    GB2312[3982]:= 16#f1b6;
    GB2312[3983]:= 16#f1b7;
    GB2312[3984]:= 16#bfd5;
    GB2312[3985]:= 16#b4a9;
    GB2312[3986]:= 16#f1b8;
    GB2312[3987]:= 16#cdbb;
    GB2312[3988]:= 16#c7d4;
    GB2312[3989]:= 16#d5ad;
    GB2312[3990]:= 16#f1b9;
    GB2312[3991]:= 16#f1ba;
    GB2312[3992]:= 16#c7cf;
    GB2312[3993]:= 16#d2a4;
    GB2312[3994]:= 16#d6cf;
    GB2312[3995]:= 16#f1bb;
    GB2312[3996]:= 16#bdd1;
    GB2312[3997]:= 16#b4b0;
    GB2312[3998]:= 16#bebd;
    GB2312[3999]:= 16#b4dc;              //GB2312码 3000-3999
END_IF;
(* Rung 15 *)
IF P_On THEN
    GB2312[4000]:= 16#ced1;
    GB2312[4001]:= 16#bfdf;
    GB2312[4002]:= 16#f1bd;
    GB2312[4003]:= 16#bffa;
    GB2312[4004]:= 16#f1bc;
    GB2312[4005]:= 16#f1bf;
    GB2312[4006]:= 16#f1be;
    GB2312[4007]:= 16#f1c0;
    GB2312[4008]:= 16#f1c1;
    GB2312[4009]:= 16#c1fe;
    GB2312[4010]:= 16#c1a2;
    GB2312[4011]:= 16#cafa;
    GB2312[4012]:= 16#d5be;
    GB2312[4013]:= 16#beba;
    GB2312[4014]:= 16#beb9;
    GB2312[4015]:= 16#d5c2;
    GB2312[4016]:= 16#bfa2;
    GB2312[4017]:= 16#cdaf;
    GB2312[4018]:= 16#f1b5;
    GB2312[4019]:= 16#bddf;
    GB2312[4020]:= 16#b6cb;
    GB2312[4021]:= 16#d6f1;
    GB2312[4022]:= 16#f3c3;
    GB2312[4023]:= 16#f3c4;
    GB2312[4024]:= 16#b8cd;
    GB2312[4025]:= 16#f3c6;
    GB2312[4026]:= 16#f3c7;
    GB2312[4027]:= 16#b0ca;
    GB2312[4028]:= 16#f3c5;
    GB2312[4029]:= 16#f3c9;
    GB2312[4030]:= 16#cbf1;
    GB2312[4031]:= 16#f3cb;
    GB2312[4032]:= 16#d0a6;
    GB2312[4033]:= 16#b1ca;
    GB2312[4034]:= 16#f3c8;
    GB2312[4035]:= 16#f3cf;
    GB2312[4036]:= 16#b5d1;
    GB2312[4037]:= 16#f3d7;
    GB2312[4038]:= 16#f3d2;
    GB2312[4039]:= 16#f3d4;
    GB2312[4040]:= 16#f3d3;
    GB2312[4041]:= 16#b7fb;
    GB2312[4042]:= 16#b1bf;
    GB2312[4043]:= 16#f3ce;
    GB2312[4044]:= 16#f3ca;
    GB2312[4045]:= 16#b5da;
    GB2312[4046]:= 16#f3d0;
    GB2312[4047]:= 16#f3d1;
    GB2312[4048]:= 16#f3d5;
    GB2312[4049]:= 16#f3cd;
    GB2312[4050]:= 16#bce3;
    GB2312[4051]:= 16#c1fd;
    GB2312[4052]:= 16#f3d6;
    GB2312[4053]:= 16#f3da;
    GB2312[4054]:= 16#f3cc;
    GB2312[4055]:= 16#b5c8;
    GB2312[4056]:= 16#bdee;
    GB2312[4057]:= 16#f3dc;
    GB2312[4058]:= 16#b7a4;
    GB2312[4059]:= 16#bff0;
    GB2312[4060]:= 16#d6fe;
    GB2312[4061]:= 16#cdb2;
    GB2312[4062]:= 16#b4f0;
    GB2312[4063]:= 16#b2df;
    GB2312[4064]:= 16#f3d8;
    GB2312[4065]:= 16#f3d9;
    GB2312[4066]:= 16#c9b8;
    GB2312[4067]:= 16#f3dd;
    GB2312[4068]:= 16#f3de;
    GB2312[4069]:= 16#f3e1;
    GB2312[4070]:= 16#f3df;
    GB2312[4071]:= 16#f3e3;
    GB2312[4072]:= 16#f3e2;
    GB2312[4073]:= 16#f3db;
    GB2312[4074]:= 16#bfea;
    GB2312[4075]:= 16#b3ef;
    GB2312[4076]:= 16#f3e0;
    GB2312[4077]:= 16#c7a9;
    GB2312[4078]:= 16#bcf2;
    GB2312[4079]:= 16#f3eb;
    GB2312[4080]:= 16#b9bf;
    GB2312[4081]:= 16#f3e4;
    GB2312[4082]:= 16#b2ad;
    GB2312[4083]:= 16#bbfe;
    GB2312[4084]:= 16#cbe3;
    GB2312[4085]:= 16#f3ed;
    GB2312[4086]:= 16#f3e9;
    GB2312[4087]:= 16#b9dc;
    GB2312[4088]:= 16#f3ee;
    GB2312[4089]:= 16#f3e5;
    GB2312[4090]:= 16#f3e6;
    GB2312[4091]:= 16#f3ea;
    GB2312[4092]:= 16#c2e1;
    GB2312[4093]:= 16#f3ec;
    GB2312[4094]:= 16#f3ef;
    GB2312[4095]:= 16#f3e8;
    GB2312[4096]:= 16#bcfd;
    GB2312[4097]:= 16#cfe4;
    GB2312[4098]:= 16#f3f0;
    GB2312[4099]:= 16#f3e7;
    GB2312[4100]:= 16#f3f2;
    GB2312[4101]:= 16#d7ad;
    GB2312[4102]:= 16#c6aa;
    GB2312[4103]:= 16#f3f3;
    GB2312[4104]:= 16#f3f1;
    GB2312[4105]:= 16#c2a8;
    GB2312[4106]:= 16#b8dd;
    GB2312[4107]:= 16#f3f5;
    GB2312[4108]:= 16#f3f4;
    GB2312[4109]:= 16#b4db;
    GB2312[4110]:= 16#f3f6;
    GB2312[4111]:= 16#f3f7;
    GB2312[4112]:= 16#f3f8;
    GB2312[4113]:= 16#c0ba;
    GB2312[4114]:= 16#c0e9;
    GB2312[4115]:= 16#c5f1;
    GB2312[4116]:= 16#f3fb;
    GB2312[4117]:= 16#f3fa;
    GB2312[4118]:= 16#b4d8;
    GB2312[4119]:= 16#f3fe;
    GB2312[4120]:= 16#f3f9;
    GB2312[4121]:= 16#f3fc;
    GB2312[4122]:= 16#f3fd;
    GB2312[4123]:= 16#f4a1;
    GB2312[4124]:= 16#f4a3;
    GB2312[4125]:= 16#bbc9;
    GB2312[4126]:= 16#f4a2;
    GB2312[4127]:= 16#f4a4;
    GB2312[4128]:= 16#b2be;
    GB2312[4129]:= 16#f4a6;
    GB2312[4130]:= 16#f4a5;
    GB2312[4131]:= 16#bcae;
    GB2312[4132]:= 16#c3d7;
    GB2312[4133]:= 16#d9e1;
    GB2312[4134]:= 16#c0e0;
    GB2312[4135]:= 16#f4cc;
    GB2312[4136]:= 16#d7d1;
    GB2312[4137]:= 16#b7db;
    GB2312[4138]:= 16#f4ce;
    GB2312[4139]:= 16#c1a3;
    GB2312[4140]:= 16#c6c9;
    GB2312[4141]:= 16#b4d6;
    GB2312[4142]:= 16#d5b3;
    GB2312[4143]:= 16#f4d0;
    GB2312[4144]:= 16#f4cf;
    GB2312[4145]:= 16#f4d1;
    GB2312[4146]:= 16#cbda;
    GB2312[4147]:= 16#f4d2;
    GB2312[4148]:= 16#d4c1;
    GB2312[4149]:= 16#d6e0;
    GB2312[4150]:= 16#b7e0;
    GB2312[4151]:= 16#c1b8;
    GB2312[4152]:= 16#c1bb;
    GB2312[4153]:= 16#f4d3;
    GB2312[4154]:= 16#beac;
    GB2312[4155]:= 16#b4e2;
    GB2312[4156]:= 16#f4d4;
    GB2312[4157]:= 16#f4d5;
    GB2312[4158]:= 16#beab;
    GB2312[4159]:= 16#f4d6;
    GB2312[4160]:= 16#f4db;
    GB2312[4161]:= 16#f4d7;
    GB2312[4162]:= 16#f4da;
    GB2312[4163]:= 16#bafd;
    GB2312[4164]:= 16#f4d8;
    GB2312[4165]:= 16#f4d9;
    GB2312[4166]:= 16#b8e2;
    GB2312[4167]:= 16#ccc7;
    GB2312[4168]:= 16#f4dc;
    GB2312[4169]:= 16#b2da;
    GB2312[4170]:= 16#c3d3;
    GB2312[4171]:= 16#d4e3;
    GB2312[4172]:= 16#bfb7;
    GB2312[4173]:= 16#f4dd;
    GB2312[4174]:= 16#c5b4;
    GB2312[4175]:= 16#f4e9;
    GB2312[4176]:= 16#cfb5;
    GB2312[4177]:= 16#cec9;
    GB2312[4178]:= 16#cbd8;
    GB2312[4179]:= 16#cbf7;
    GB2312[4180]:= 16#bdf4;
    GB2312[4181]:= 16#d7cf;
    GB2312[4182]:= 16#c0db;
    GB2312[4183]:= 16#d0f5;
    GB2312[4184]:= 16#f4ea;
    GB2312[4185]:= 16#f4eb;
    GB2312[4186]:= 16#f4ec;
    GB2312[4187]:= 16#f7e3;
    GB2312[4188]:= 16#b7b1;
    GB2312[4189]:= 16#f4ed;
    GB2312[4190]:= 16#d7eb;
    GB2312[4191]:= 16#f4ee;
    GB2312[4192]:= 16#e6f9;
    GB2312[4193]:= 16#bec0;
    GB2312[4194]:= 16#e6fa;
    GB2312[4195]:= 16#baec;
    GB2312[4196]:= 16#e6fb;
    GB2312[4197]:= 16#cfcb;
    GB2312[4198]:= 16#e6fc;
    GB2312[4199]:= 16#d4bc;
    GB2312[4200]:= 16#bcb6;
    GB2312[4201]:= 16#e6fd;
    GB2312[4202]:= 16#e6fe;
    GB2312[4203]:= 16#bccd;
    GB2312[4204]:= 16#c8d2;
    GB2312[4205]:= 16#ceb3;
    GB2312[4206]:= 16#e7a1;
    GB2312[4207]:= 16#b4bf;
    GB2312[4208]:= 16#e7a2;
    GB2312[4209]:= 16#c9b4;
    GB2312[4210]:= 16#b8d9;
    GB2312[4211]:= 16#c4c9;
    GB2312[4212]:= 16#d7dd;
    GB2312[4213]:= 16#c2da;
    GB2312[4214]:= 16#b7d7;
    GB2312[4215]:= 16#d6bd;
    GB2312[4216]:= 16#cec6;
    GB2312[4217]:= 16#b7c4;
    GB2312[4218]:= 16#c5a6;
    GB2312[4219]:= 16#e7a3;
    GB2312[4220]:= 16#cfdf;
    GB2312[4221]:= 16#e7a4;
    GB2312[4222]:= 16#e7a5;
    GB2312[4223]:= 16#e7a6;
    GB2312[4224]:= 16#c1b7;
    GB2312[4225]:= 16#d7e9;
    GB2312[4226]:= 16#c9f0;
    GB2312[4227]:= 16#cfb8;
    GB2312[4228]:= 16#d6af;
    GB2312[4229]:= 16#d6d5;
    GB2312[4230]:= 16#e7a7;
    GB2312[4231]:= 16#b0ed;
    GB2312[4232]:= 16#e7a8;
    GB2312[4233]:= 16#e7a9;
    GB2312[4234]:= 16#c9dc;
    GB2312[4235]:= 16#d2ef;
    GB2312[4236]:= 16#bead;
    GB2312[4237]:= 16#e7aa;
    GB2312[4238]:= 16#b0f3;
    GB2312[4239]:= 16#c8de;
    GB2312[4240]:= 16#bde1;
    GB2312[4241]:= 16#e7ab;
    GB2312[4242]:= 16#c8c6;
    GB2312[4243]:= 16#e7ac;
    GB2312[4244]:= 16#bbe6;
    GB2312[4245]:= 16#b8f8;
    GB2312[4246]:= 16#d1a4;
    GB2312[4247]:= 16#e7ad;
    GB2312[4248]:= 16#c2e7;
    GB2312[4249]:= 16#bef8;
    GB2312[4250]:= 16#bdca;
    GB2312[4251]:= 16#cdb3;
    GB2312[4252]:= 16#e7ae;
    GB2312[4253]:= 16#e7af;
    GB2312[4254]:= 16#beee;
    GB2312[4255]:= 16#d0e5;
    GB2312[4256]:= 16#cbe7;
    GB2312[4257]:= 16#ccd0;
    GB2312[4258]:= 16#bccc;
    GB2312[4259]:= 16#e7b0;
    GB2312[4260]:= 16#bca8;
    GB2312[4261]:= 16#d0f7;
    GB2312[4262]:= 16#e7b1;
    GB2312[4263]:= 16#d0f8;
    GB2312[4264]:= 16#e7b2;
    GB2312[4265]:= 16#e7b3;
    GB2312[4266]:= 16#b4c2;
    GB2312[4267]:= 16#e7b4;
    GB2312[4268]:= 16#e7b5;
    GB2312[4269]:= 16#c9fe;
    GB2312[4270]:= 16#ceac;
    GB2312[4271]:= 16#c3e0;
    GB2312[4272]:= 16#e7b7;
    GB2312[4273]:= 16#b1c1;
    GB2312[4274]:= 16#b3f1;
    GB2312[4275]:= 16#e7b8;
    GB2312[4276]:= 16#e7b9;
    GB2312[4277]:= 16#d7db;
    GB2312[4278]:= 16#d5c0;
    GB2312[4279]:= 16#e7ba;
    GB2312[4280]:= 16#c2cc;
    GB2312[4281]:= 16#d7ba;
    GB2312[4282]:= 16#e7bb;
    GB2312[4283]:= 16#e7bc;
    GB2312[4284]:= 16#e7bd;
    GB2312[4285]:= 16#bcea;
    GB2312[4286]:= 16#c3e5;
    GB2312[4287]:= 16#c0c2;
    GB2312[4288]:= 16#e7be;
    GB2312[4289]:= 16#e7bf;
    GB2312[4290]:= 16#bca9;
    GB2312[4291]:= 16#e7c0;
    GB2312[4292]:= 16#e7c1;
    GB2312[4293]:= 16#e7b6;
    GB2312[4294]:= 16#b6d0;
    GB2312[4295]:= 16#e7c2;
    GB2312[4296]:= 16#e7c3;
    GB2312[4297]:= 16#e7c4;
    GB2312[4298]:= 16#bbba;
    GB2312[4299]:= 16#b5de;
    GB2312[4300]:= 16#c2c6;
    GB2312[4301]:= 16#b1e0;
    GB2312[4302]:= 16#e7c5;
    GB2312[4303]:= 16#d4b5;
    GB2312[4304]:= 16#e7c6;
    GB2312[4305]:= 16#b8bf;
    GB2312[4306]:= 16#e7c8;
    GB2312[4307]:= 16#e7c7;
    GB2312[4308]:= 16#b7ec;
    GB2312[4309]:= 16#e7c9;
    GB2312[4310]:= 16#b2f8;
    GB2312[4311]:= 16#e7ca;
    GB2312[4312]:= 16#e7cb;
    GB2312[4313]:= 16#e7cc;
    GB2312[4314]:= 16#e7cd;
    GB2312[4315]:= 16#e7ce;
    GB2312[4316]:= 16#e7cf;
    GB2312[4317]:= 16#e7d0;
    GB2312[4318]:= 16#d3a7;
    GB2312[4319]:= 16#cbf5;
    GB2312[4320]:= 16#e7d1;
    GB2312[4321]:= 16#e7d2;
    GB2312[4322]:= 16#e7d3;
    GB2312[4323]:= 16#e7d4;
    GB2312[4324]:= 16#c9c9;
    GB2312[4325]:= 16#e7d5;
    GB2312[4326]:= 16#e7d6;
    GB2312[4327]:= 16#e7d7;
    GB2312[4328]:= 16#e7d8;
    GB2312[4329]:= 16#e7d9;
    GB2312[4330]:= 16#bdc9;
    GB2312[4331]:= 16#e7da;
    GB2312[4332]:= 16#f3be;
    GB2312[4333]:= 16#b8d7;
    GB2312[4334]:= 16#c8b1;
    GB2312[4335]:= 16#f3bf;
    GB2312[4336]:= 16#f3c0;
    GB2312[4337]:= 16#f3c1;
    GB2312[4338]:= 16#b9de;
    GB2312[4339]:= 16#cdf8;
    GB2312[4340]:= 16#d8e8;
    GB2312[4341]:= 16#bab1;
    GB2312[4342]:= 16#c2de;
    GB2312[4343]:= 16#eeb7;
    GB2312[4344]:= 16#b7a3;
    GB2312[4345]:= 16#eeb9;
    GB2312[4346]:= 16#eeb8;
    GB2312[4347]:= 16#b0d5;
    GB2312[4348]:= 16#eebb;
    GB2312[4349]:= 16#d5d6;
    GB2312[4350]:= 16#d7ef;
    GB2312[4351]:= 16#d6c3;
    GB2312[4352]:= 16#eebd;
    GB2312[4353]:= 16#caf0;
    GB2312[4354]:= 16#eebc;
    GB2312[4355]:= 16#eebe;
    GB2312[4356]:= 16#eec0;
    GB2312[4357]:= 16#eebf;
    GB2312[4358]:= 16#d1f2;
    GB2312[4359]:= 16#c7bc;
    GB2312[4360]:= 16#c3c0;
    GB2312[4361]:= 16#b8e1;
    GB2312[4362]:= 16#c1e7;
    GB2312[4363]:= 16#f4c6;
    GB2312[4364]:= 16#d0df;
    GB2312[4365]:= 16#f4c7;
    GB2312[4366]:= 16#cfdb;
    GB2312[4367]:= 16#c8ba;
    GB2312[4368]:= 16#f4c8;
    GB2312[4369]:= 16#f4c9;
    GB2312[4370]:= 16#f4ca;
    GB2312[4371]:= 16#f4cb;
    GB2312[4372]:= 16#d9fa;
    GB2312[4373]:= 16#b8fe;
    GB2312[4374]:= 16#e5f1;
    GB2312[4375]:= 16#d3f0;
    GB2312[4376]:= 16#f4e0;
    GB2312[4377]:= 16#cecc;
    GB2312[4378]:= 16#b3e1;
    GB2312[4379]:= 16#f1b4;
    GB2312[4380]:= 16#d2ee;
    GB2312[4381]:= 16#f4e1;
    GB2312[4382]:= 16#cfe8;
    GB2312[4383]:= 16#f4e2;
    GB2312[4384]:= 16#c7cc;
    GB2312[4385]:= 16#b5d4;
    GB2312[4386]:= 16#b4e4;
    GB2312[4387]:= 16#f4e4;
    GB2312[4388]:= 16#f4e3;
    GB2312[4389]:= 16#f4e5;
    GB2312[4390]:= 16#f4e6;
    GB2312[4391]:= 16#f4e7;
    GB2312[4392]:= 16#bab2;
    GB2312[4393]:= 16#b0bf;
    GB2312[4394]:= 16#f4e8;
    GB2312[4395]:= 16#b7ad;
    GB2312[4396]:= 16#d2ed;
    GB2312[4397]:= 16#d2ab;
    GB2312[4398]:= 16#c0cf;
    GB2312[4399]:= 16#bfbc;
    GB2312[4400]:= 16#eba3;
    GB2312[4401]:= 16#d5df;
    GB2312[4402]:= 16#eac8;
    GB2312[4403]:= 16#f1f3;
    GB2312[4404]:= 16#b6f8;
    GB2312[4405]:= 16#cba3;
    GB2312[4406]:= 16#c4cd;
    GB2312[4407]:= 16#f1e7;
    GB2312[4408]:= 16#f1e8;
    GB2312[4409]:= 16#b8fb;
    GB2312[4410]:= 16#f1e9;
    GB2312[4411]:= 16#bac4;
    GB2312[4412]:= 16#d4c5;
    GB2312[4413]:= 16#b0d2;
    GB2312[4414]:= 16#f1ea;
    GB2312[4415]:= 16#f1eb;
    GB2312[4416]:= 16#f1ec;
    GB2312[4417]:= 16#f1ed;
    GB2312[4418]:= 16#f1ee;
    GB2312[4419]:= 16#f1ef;
    GB2312[4420]:= 16#f1f1;
    GB2312[4421]:= 16#f1f0;
    GB2312[4422]:= 16#c5d5;
    GB2312[4423]:= 16#f1f2;
    GB2312[4424]:= 16#b6fa;
    GB2312[4425]:= 16#f1f4;
    GB2312[4426]:= 16#d2ae;
    GB2312[4427]:= 16#dec7;
    GB2312[4428]:= 16#cbca;
    GB2312[4429]:= 16#b3dc;
    GB2312[4430]:= 16#b5a2;
    GB2312[4431]:= 16#b9a2;
    GB2312[4432]:= 16#c4f4;
    GB2312[4433]:= 16#f1f5;
    GB2312[4434]:= 16#f1f6;
    GB2312[4435]:= 16#c1c4;
    GB2312[4436]:= 16#c1fb;
    GB2312[4437]:= 16#d6b0;
    GB2312[4438]:= 16#f1f7;
    GB2312[4439]:= 16#f1f8;
    GB2312[4440]:= 16#c1aa;
    GB2312[4441]:= 16#c6b8;
    GB2312[4442]:= 16#bedb;
    GB2312[4443]:= 16#f1f9;
    GB2312[4444]:= 16#b4cf;
    GB2312[4445]:= 16#f1fa;
    GB2312[4446]:= 16#edb2;
    GB2312[4447]:= 16#edb1;
    GB2312[4448]:= 16#cbe0;
    GB2312[4449]:= 16#d2de;
    GB2312[4450]:= 16#cbc1;
    GB2312[4451]:= 16#d5d8;
    GB2312[4452]:= 16#c8e2;
    GB2312[4453]:= 16#c0df;
    GB2312[4454]:= 16#bca1;
    GB2312[4455]:= 16#ebc1;
    GB2312[4456]:= 16#d0a4;
    GB2312[4457]:= 16#d6e2;
    GB2312[4458]:= 16#b6c7;
    GB2312[4459]:= 16#b8d8;
    GB2312[4460]:= 16#ebc0;
    GB2312[4461]:= 16#b8ce;
    GB2312[4462]:= 16#ebbf;
    GB2312[4463]:= 16#b3a6;
    GB2312[4464]:= 16#b9c9;
    GB2312[4465]:= 16#d6ab;
    GB2312[4466]:= 16#b7f4;
    GB2312[4467]:= 16#b7ca;
    GB2312[4468]:= 16#bce7;
    GB2312[4469]:= 16#b7be;
    GB2312[4470]:= 16#ebc6;
    GB2312[4471]:= 16#ebc7;
    GB2312[4472]:= 16#b0b9;
    GB2312[4473]:= 16#bfcf;
    GB2312[4474]:= 16#ebc5;
    GB2312[4475]:= 16#d3fd;
    GB2312[4476]:= 16#ebc8;
    GB2312[4477]:= 16#ebc9;
    GB2312[4478]:= 16#b7ce;
    GB2312[4479]:= 16#ebc2;
    GB2312[4480]:= 16#ebc4;
    GB2312[4481]:= 16#c9f6;
    GB2312[4482]:= 16#d6d7;
    GB2312[4483]:= 16#d5cd;
    GB2312[4484]:= 16#d0b2;
    GB2312[4485]:= 16#ebcf;
    GB2312[4486]:= 16#ceb8;
    GB2312[4487]:= 16#ebd0;
    GB2312[4488]:= 16#b5a8;
    GB2312[4489]:= 16#b1b3;
    GB2312[4490]:= 16#ebd2;
    GB2312[4491]:= 16#cca5;
    GB2312[4492]:= 16#c5d6;
    GB2312[4493]:= 16#ebd3;
    GB2312[4494]:= 16#ebd1;
    GB2312[4495]:= 16#c5df;
    GB2312[4496]:= 16#ebce;
    GB2312[4497]:= 16#caa4;
    GB2312[4498]:= 16#ebd5;
    GB2312[4499]:= 16#b0fb;
    GB2312[4500]:= 16#bafa;
    GB2312[4501]:= 16#d8b7;
    GB2312[4502]:= 16#f1e3;
    GB2312[4503]:= 16#ebca;
    GB2312[4504]:= 16#ebcb;
    GB2312[4505]:= 16#ebcc;
    GB2312[4506]:= 16#ebcd;
    GB2312[4507]:= 16#ebd6;
    GB2312[4508]:= 16#e6c0;
    GB2312[4509]:= 16#ebd9;
    GB2312[4510]:= 16#bfe8;
    GB2312[4511]:= 16#d2c8;
    GB2312[4512]:= 16#ebd7;
    GB2312[4513]:= 16#ebdc;
    GB2312[4514]:= 16#b8ec;
    GB2312[4515]:= 16#ebd8;
    GB2312[4516]:= 16#bdba;
    GB2312[4517]:= 16#d0d8;
    GB2312[4518]:= 16#b0b7;
    GB2312[4519]:= 16#ebdd;
    GB2312[4520]:= 16#c4dc;
    GB2312[4521]:= 16#d6ac;
    GB2312[4522]:= 16#b4e0;
    GB2312[4523]:= 16#c2f6;
    GB2312[4524]:= 16#bcb9;
    GB2312[4525]:= 16#ebda;
    GB2312[4526]:= 16#ebdb;
    GB2312[4527]:= 16#d4e0;
    GB2312[4528]:= 16#c6ea;
    GB2312[4529]:= 16#c4d4;
    GB2312[4530]:= 16#ebdf;
    GB2312[4531]:= 16#c5a7;
    GB2312[4532]:= 16#d9f5;
    GB2312[4533]:= 16#b2b1;
    GB2312[4534]:= 16#ebe4;
    GB2312[4535]:= 16#bdc5;
    GB2312[4536]:= 16#ebe2;
    GB2312[4537]:= 16#ebe3;
    GB2312[4538]:= 16#b8ac;
    GB2312[4539]:= 16#cdd1;
    GB2312[4540]:= 16#ebe5;
    GB2312[4541]:= 16#ebe1;
    GB2312[4542]:= 16#c1b3;
    GB2312[4543]:= 16#c6a2;
    GB2312[4544]:= 16#ccf3;
    GB2312[4545]:= 16#ebe6;
    GB2312[4546]:= 16#c0b0;
    GB2312[4547]:= 16#d2b8;
    GB2312[4548]:= 16#ebe7;
    GB2312[4549]:= 16#b8af;
    GB2312[4550]:= 16#b8ad;
    GB2312[4551]:= 16#ebe8;
    GB2312[4552]:= 16#c7bb;
    GB2312[4553]:= 16#cdf3;
    GB2312[4554]:= 16#ebea;
    GB2312[4555]:= 16#ebeb;
    GB2312[4556]:= 16#ebed;
    GB2312[4557]:= 16#d0c8;
    GB2312[4558]:= 16#ebf2;
    GB2312[4559]:= 16#ebee;
    GB2312[4560]:= 16#ebf1;
    GB2312[4561]:= 16#c8f9;
    GB2312[4562]:= 16#d1fc;
    GB2312[4563]:= 16#ebec;
    GB2312[4564]:= 16#ebe9;
    GB2312[4565]:= 16#b8b9;
    GB2312[4566]:= 16#cfd9;
    GB2312[4567]:= 16#c4e5;
    GB2312[4568]:= 16#ebef;
    GB2312[4569]:= 16#ebf0;
    GB2312[4570]:= 16#ccda;
    GB2312[4571]:= 16#cdc8;
    GB2312[4572]:= 16#b0f2;
    GB2312[4573]:= 16#ebf6;
    GB2312[4574]:= 16#ebf5;
    GB2312[4575]:= 16#b2b2;
    GB2312[4576]:= 16#b8e0;
    GB2312[4577]:= 16#ebf7;
    GB2312[4578]:= 16#b1ec;
    GB2312[4579]:= 16#ccc5;
    GB2312[4580]:= 16#c4a4;
    GB2312[4581]:= 16#cfa5;
    GB2312[4582]:= 16#ebf9;
    GB2312[4583]:= 16#eca2;
    GB2312[4584]:= 16#c5f2;
    GB2312[4585]:= 16#ebfa;
    GB2312[4586]:= 16#c9c5;
    GB2312[4587]:= 16#e2df;
    GB2312[4588]:= 16#ebfe;
    GB2312[4589]:= 16#cdce;
    GB2312[4590]:= 16#eca1;
    GB2312[4591]:= 16#b1db;
    GB2312[4592]:= 16#d3b7;
    GB2312[4593]:= 16#d2dc;
    GB2312[4594]:= 16#ebfd;
    GB2312[4595]:= 16#ebfb;
    GB2312[4596]:= 16#b3bc;
    GB2312[4597]:= 16#eab0;
    GB2312[4598]:= 16#d7d4;
    GB2312[4599]:= 16#f4ab;
    GB2312[4600]:= 16#b3f4;
    GB2312[4601]:= 16#d6c1;
    GB2312[4602]:= 16#d6c2;
    GB2312[4603]:= 16#d5e9;
    GB2312[4604]:= 16#beca;
    GB2312[4605]:= 16#f4a7;
    GB2312[4606]:= 16#d2a8;
    GB2312[4607]:= 16#f4a8;
    GB2312[4608]:= 16#f4a9;
    GB2312[4609]:= 16#f4aa;
    GB2312[4610]:= 16#becb;
    GB2312[4611]:= 16#d3df;
    GB2312[4612]:= 16#c9e0;
    GB2312[4613]:= 16#c9e1;
    GB2312[4614]:= 16#f3c2;
    GB2312[4615]:= 16#cae6;
    GB2312[4616]:= 16#ccf2;
    GB2312[4617]:= 16#e2b6;
    GB2312[4618]:= 16#cbb4;
    GB2312[4619]:= 16#cee8;
    GB2312[4620]:= 16#d6db;
    GB2312[4621]:= 16#f4ad;
    GB2312[4622]:= 16#f4ae;
    GB2312[4623]:= 16#f4af;
    GB2312[4624]:= 16#f4b2;
    GB2312[4625]:= 16#babd;
    GB2312[4626]:= 16#f4b3;
    GB2312[4627]:= 16#b0e3;
    GB2312[4628]:= 16#f4b0;
    GB2312[4629]:= 16#f4b1;
    GB2312[4630]:= 16#bda2;
    GB2312[4631]:= 16#b2d5;
    GB2312[4632]:= 16#f4b6;
    GB2312[4633]:= 16#f4b7;
    GB2312[4634]:= 16#b6e6;
    GB2312[4635]:= 16#b2b0;
    GB2312[4636]:= 16#cfcf;
    GB2312[4637]:= 16#f4b4;
    GB2312[4638]:= 16#b4ac;
    GB2312[4639]:= 16#f4b5;
    GB2312[4640]:= 16#f4b8;
    GB2312[4641]:= 16#f4b9;
    GB2312[4642]:= 16#cda7;
    GB2312[4643]:= 16#f4ba;
    GB2312[4644]:= 16#f4bb;
    GB2312[4645]:= 16#f4bc;
    GB2312[4646]:= 16#cbd2;
    GB2312[4647]:= 16#f4bd;
    GB2312[4648]:= 16#f4be;
    GB2312[4649]:= 16#f4bf;
    GB2312[4650]:= 16#f4de;
    GB2312[4651]:= 16#c1bc;
    GB2312[4652]:= 16#bce8;
    GB2312[4653]:= 16#c9ab;
    GB2312[4654]:= 16#d1de;
    GB2312[4655]:= 16#e5f5;
    GB2312[4656]:= 16#dcb3;
    GB2312[4657]:= 16#d2d5;
    GB2312[4658]:= 16#dcb4;
    GB2312[4659]:= 16#b0ac;
    GB2312[4660]:= 16#dcb5;
    GB2312[4661]:= 16#bdda;
    GB2312[4662]:= 16#dcb9;
    GB2312[4663]:= 16#d8c2;
    GB2312[4664]:= 16#dcb7;
    GB2312[4665]:= 16#d3f3;
    GB2312[4666]:= 16#c9d6;
    GB2312[4667]:= 16#dcba;
    GB2312[4668]:= 16#dcb6;
    GB2312[4669]:= 16#dcbb;
    GB2312[4670]:= 16#c3a2;
    GB2312[4671]:= 16#dcbc;
    GB2312[4672]:= 16#dcc5;
    GB2312[4673]:= 16#dcbd;
    GB2312[4674]:= 16#cedf;
    GB2312[4675]:= 16#d6a5;
    GB2312[4676]:= 16#dccf;
    GB2312[4677]:= 16#dccd;
    GB2312[4678]:= 16#dcd2;
    GB2312[4679]:= 16#bde6;
    GB2312[4680]:= 16#c2ab;
    GB2312[4681]:= 16#dcb8;
    GB2312[4682]:= 16#dccb;
    GB2312[4683]:= 16#dcce;
    GB2312[4684]:= 16#dcbe;
    GB2312[4685]:= 16#b7d2;
    GB2312[4686]:= 16#b0c5;
    GB2312[4687]:= 16#dcc7;
    GB2312[4688]:= 16#d0be;
    GB2312[4689]:= 16#dcc1;
    GB2312[4690]:= 16#bba8;
    GB2312[4691]:= 16#b7bc;
    GB2312[4692]:= 16#dccc;
    GB2312[4693]:= 16#dcc6;
    GB2312[4694]:= 16#dcbf;
    GB2312[4695]:= 16#c7db;
    GB2312[4696]:= 16#d1bf;
    GB2312[4697]:= 16#dcc0;
    GB2312[4698]:= 16#dcca;
    GB2312[4699]:= 16#dcd0;
    GB2312[4700]:= 16#cead;
    GB2312[4701]:= 16#dcc2;
    GB2312[4702]:= 16#dcc3;
    GB2312[4703]:= 16#dcc8;
    GB2312[4704]:= 16#dcc9;
    GB2312[4705]:= 16#b2d4;
    GB2312[4706]:= 16#dcd1;
    GB2312[4707]:= 16#cbd5;
    GB2312[4708]:= 16#d4b7;
    GB2312[4709]:= 16#dcdb;
    GB2312[4710]:= 16#dcdf;
    GB2312[4711]:= 16#cca6;
    GB2312[4712]:= 16#dce6;
    GB2312[4713]:= 16#c3e7;
    GB2312[4714]:= 16#dcdc;
    GB2312[4715]:= 16#bfc1;
    GB2312[4716]:= 16#dcd9;
    GB2312[4717]:= 16#b0fa;
    GB2312[4718]:= 16#b9b6;
    GB2312[4719]:= 16#dce5;
    GB2312[4720]:= 16#dcd3;
    GB2312[4721]:= 16#dcc4;
    GB2312[4722]:= 16#dcd6;
    GB2312[4723]:= 16#c8f4;
    GB2312[4724]:= 16#bfe0;
    GB2312[4725]:= 16#c9bb;
    GB2312[4726]:= 16#b1bd;
    GB2312[4727]:= 16#d3a2;
    GB2312[4728]:= 16#dcda;
    GB2312[4729]:= 16#dcd5;
    GB2312[4730]:= 16#c6bb;
    GB2312[4731]:= 16#dcde;
    GB2312[4732]:= 16#d7c2;
    GB2312[4733]:= 16#c3af;
    GB2312[4734]:= 16#b7b6;
    GB2312[4735]:= 16#c7d1;
    GB2312[4736]:= 16#c3a9;
    GB2312[4737]:= 16#dce2;
    GB2312[4738]:= 16#dcd8;
    GB2312[4739]:= 16#dceb;
    GB2312[4740]:= 16#dcd4;
    GB2312[4741]:= 16#dcdd;
    GB2312[4742]:= 16#bea5;
    GB2312[4743]:= 16#dcd7;
    GB2312[4744]:= 16#dce0;
    GB2312[4745]:= 16#dce3;
    GB2312[4746]:= 16#dce4;
    GB2312[4747]:= 16#dcf8;
    GB2312[4748]:= 16#dce1;
    GB2312[4749]:= 16#dda2;
    GB2312[4750]:= 16#dce7;
    GB2312[4751]:= 16#bceb;
    GB2312[4752]:= 16#b4c4;
    GB2312[4753]:= 16#c3a3;
    GB2312[4754]:= 16#b2e7;
    GB2312[4755]:= 16#dcfa;
    GB2312[4756]:= 16#dcf2;
    GB2312[4757]:= 16#dcef;
    GB2312[4758]:= 16#dcfc;
    GB2312[4759]:= 16#dcee;
    GB2312[4760]:= 16#d2f0;
    GB2312[4761]:= 16#b2e8;
    GB2312[4762]:= 16#c8d7;
    GB2312[4763]:= 16#c8e3;
    GB2312[4764]:= 16#dcfb;
    GB2312[4765]:= 16#dced;
    GB2312[4766]:= 16#dcf7;
    GB2312[4767]:= 16#dcf5;
    GB2312[4768]:= 16#bea3;
    GB2312[4769]:= 16#dcf4;
    GB2312[4770]:= 16#b2dd;
    GB2312[4771]:= 16#dcf3;
    GB2312[4772]:= 16#bcf6;
    GB2312[4773]:= 16#dce8;
    GB2312[4774]:= 16#bbc4;
    GB2312[4775]:= 16#c0f3;
    GB2312[4776]:= 16#bcd4;
    GB2312[4777]:= 16#dce9;
    GB2312[4778]:= 16#dcea;
    GB2312[4779]:= 16#dcf1;
    GB2312[4780]:= 16#dcf6;
    GB2312[4781]:= 16#dcf9;
    GB2312[4782]:= 16#b5b4;
    GB2312[4783]:= 16#c8d9;
    GB2312[4784]:= 16#bbe7;
    GB2312[4785]:= 16#dcfe;
    GB2312[4786]:= 16#dcfd;
    GB2312[4787]:= 16#d3ab;
    GB2312[4788]:= 16#dda1;
    GB2312[4789]:= 16#dda3;
    GB2312[4790]:= 16#dda5;
    GB2312[4791]:= 16#d2f1;
    GB2312[4792]:= 16#dda4;
    GB2312[4793]:= 16#dda6;
    GB2312[4794]:= 16#dda7;
    GB2312[4795]:= 16#d2a9;
    GB2312[4796]:= 16#bac9;
    GB2312[4797]:= 16#dda9;
    GB2312[4798]:= 16#ddb6;
    GB2312[4799]:= 16#ddb1;
    GB2312[4800]:= 16#ddb4;
    GB2312[4801]:= 16#ddb0;
    GB2312[4802]:= 16#c6ce;
    GB2312[4803]:= 16#c0f2;
    GB2312[4804]:= 16#c9af;
    GB2312[4805]:= 16#dcec;
    GB2312[4806]:= 16#ddae;
    GB2312[4807]:= 16#ddb7;
    GB2312[4808]:= 16#dcf0;
    GB2312[4809]:= 16#ddaf;
    GB2312[4810]:= 16#ddb8;
    GB2312[4811]:= 16#ddac;
    GB2312[4812]:= 16#ddb9;
    GB2312[4813]:= 16#ddb3;
    GB2312[4814]:= 16#ddad;
    GB2312[4815]:= 16#c4aa;
    GB2312[4816]:= 16#dda8;
    GB2312[4817]:= 16#c0b3;
    GB2312[4818]:= 16#c1ab;
    GB2312[4819]:= 16#ddaa;
    GB2312[4820]:= 16#ddab;
    GB2312[4821]:= 16#ddb2;
    GB2312[4822]:= 16#bbf1;
    GB2312[4823]:= 16#ddb5;
    GB2312[4824]:= 16#d3a8;
    GB2312[4825]:= 16#ddba;
    GB2312[4826]:= 16#ddbb;
    GB2312[4827]:= 16#c3a7;
    GB2312[4828]:= 16#ddd2;
    GB2312[4829]:= 16#ddbc;
    GB2312[4830]:= 16#ddd1;
    GB2312[4831]:= 16#b9bd;
    GB2312[4832]:= 16#bed5;
    GB2312[4833]:= 16#befa;
    GB2312[4834]:= 16#baca;
    GB2312[4835]:= 16#ddca;
    GB2312[4836]:= 16#ddc5;
    GB2312[4837]:= 16#ddbf;
    GB2312[4838]:= 16#b2cb;
    GB2312[4839]:= 16#ddc3;
    GB2312[4840]:= 16#ddcb;
    GB2312[4841]:= 16#b2a4;
    GB2312[4842]:= 16#ddd5;
    GB2312[4843]:= 16#ddbe;
    GB2312[4844]:= 16#c6d0;
    GB2312[4845]:= 16#ddd0;
    GB2312[4846]:= 16#ddd4;
    GB2312[4847]:= 16#c1e2;
    GB2312[4848]:= 16#b7c6;
    GB2312[4849]:= 16#ddce;
    GB2312[4850]:= 16#ddcf;
    GB2312[4851]:= 16#ddc4;
    GB2312[4852]:= 16#ddbd;
    GB2312[4853]:= 16#ddcd;
    GB2312[4854]:= 16#ccd1;
    GB2312[4855]:= 16#ddc9;
    GB2312[4856]:= 16#ddc2;
    GB2312[4857]:= 16#c3c8;
    GB2312[4858]:= 16#c6bc;
    GB2312[4859]:= 16#ceae;
    GB2312[4860]:= 16#ddcc;
    GB2312[4861]:= 16#ddc8;
    GB2312[4862]:= 16#ddc1;
    GB2312[4863]:= 16#ddc6;
    GB2312[4864]:= 16#c2dc;
    GB2312[4865]:= 16#d3a9;
    GB2312[4866]:= 16#d3aa;
    GB2312[4867]:= 16#ddd3;
    GB2312[4868]:= 16#cff4;
    GB2312[4869]:= 16#c8f8;
    GB2312[4870]:= 16#dde6;
    GB2312[4871]:= 16#ddc7;
    GB2312[4872]:= 16#dde0;
    GB2312[4873]:= 16#c2e4;
    GB2312[4874]:= 16#dde1;
    GB2312[4875]:= 16#ddd7;
    GB2312[4876]:= 16#d6f8;
    GB2312[4877]:= 16#ddd9;
    GB2312[4878]:= 16#ddd8;
    GB2312[4879]:= 16#b8f0;
    GB2312[4880]:= 16#ddd6;
    GB2312[4881]:= 16#c6cf;
    GB2312[4882]:= 16#b6ad;
    GB2312[4883]:= 16#dde2;
    GB2312[4884]:= 16#baf9;
    GB2312[4885]:= 16#d4e1;
    GB2312[4886]:= 16#dde7;
    GB2312[4887]:= 16#b4d0;
    GB2312[4888]:= 16#ddda;
    GB2312[4889]:= 16#bffb;
    GB2312[4890]:= 16#dde3;
    GB2312[4891]:= 16#dddf;
    GB2312[4892]:= 16#dddd;
    GB2312[4893]:= 16#b5d9;
    GB2312[4894]:= 16#dddb;
    GB2312[4895]:= 16#dddc;
    GB2312[4896]:= 16#ddde;
    GB2312[4897]:= 16#bdaf;
    GB2312[4898]:= 16#dde4;
    GB2312[4899]:= 16#dde5;
    GB2312[4900]:= 16#ddf5;
    GB2312[4901]:= 16#c3c9;
    GB2312[4902]:= 16#cbe2;
    GB2312[4903]:= 16#ddf2;
    GB2312[4904]:= 16#d8e1;
    GB2312[4905]:= 16#c6d1;
    GB2312[4906]:= 16#ddf4;
    GB2312[4907]:= 16#d5f4;
    GB2312[4908]:= 16#ddf3;
    GB2312[4909]:= 16#ddf0;
    GB2312[4910]:= 16#ddec;
    GB2312[4911]:= 16#ddef;
    GB2312[4912]:= 16#dde8;
    GB2312[4913]:= 16#d0ee;
    GB2312[4914]:= 16#c8d8;
    GB2312[4915]:= 16#ddee;
    GB2312[4916]:= 16#dde9;
    GB2312[4917]:= 16#ddea;
    GB2312[4918]:= 16#cbf2;
    GB2312[4919]:= 16#dded;
    GB2312[4920]:= 16#b1cd;
    GB2312[4921]:= 16#c0b6;
    GB2312[4922]:= 16#bcbb;
    GB2312[4923]:= 16#ddf1;
    GB2312[4924]:= 16#ddf7;
    GB2312[4925]:= 16#ddf6;
    GB2312[4926]:= 16#ddeb;
    GB2312[4927]:= 16#c5ee;
    GB2312[4928]:= 16#ddfb;
    GB2312[4929]:= 16#dea4;
    GB2312[4930]:= 16#dea3;
    GB2312[4931]:= 16#ddf8;
    GB2312[4932]:= 16#c3ef;
    GB2312[4933]:= 16#c2fb;
    GB2312[4934]:= 16#d5e1;
    GB2312[4935]:= 16#ceb5;
    GB2312[4936]:= 16#ddfd;
    GB2312[4937]:= 16#b2cc;
    GB2312[4938]:= 16#c4e8;
    GB2312[4939]:= 16#cadf;
    GB2312[4940]:= 16#c7be;
    GB2312[4941]:= 16#ddfa;
    GB2312[4942]:= 16#ddfc;
    GB2312[4943]:= 16#ddfe;
    GB2312[4944]:= 16#dea2;
    GB2312[4945]:= 16#b0aa;
    GB2312[4946]:= 16#b1ce;
    GB2312[4947]:= 16#deac;
    GB2312[4948]:= 16#dea6;
    GB2312[4949]:= 16#bdb6;
    GB2312[4950]:= 16#c8ef;
    GB2312[4951]:= 16#dea1;
    GB2312[4952]:= 16#dea5;
    GB2312[4953]:= 16#dea9;
    GB2312[4954]:= 16#dea8;
    GB2312[4955]:= 16#dea7;
    GB2312[4956]:= 16#dead;
    GB2312[4957]:= 16#d4cc;
    GB2312[4958]:= 16#deb3;
    GB2312[4959]:= 16#deaa;
    GB2312[4960]:= 16#deae;
    GB2312[4961]:= 16#c0d9;
    GB2312[4962]:= 16#b1a1;
    GB2312[4963]:= 16#deb6;
    GB2312[4964]:= 16#deb1;
    GB2312[4965]:= 16#deb2;
    GB2312[4966]:= 16#d1a6;
    GB2312[4967]:= 16#deb5;
    GB2312[4968]:= 16#deaf;
    GB2312[4969]:= 16#deb0;
    GB2312[4970]:= 16#d0bd;
    GB2312[4971]:= 16#deb4;
    GB2312[4972]:= 16#caed;
    GB2312[4973]:= 16#deb9;
    GB2312[4974]:= 16#deb8;
    GB2312[4975]:= 16#deb7;
    GB2312[4976]:= 16#debb;
    GB2312[4977]:= 16#bde5;
    GB2312[4978]:= 16#b2d8;
    GB2312[4979]:= 16#c3ea;
    GB2312[4980]:= 16#deba;
    GB2312[4981]:= 16#c5ba;
    GB2312[4982]:= 16#debc;
    GB2312[4983]:= 16#ccd9;
    GB2312[4984]:= 16#b7aa;
    GB2312[4985]:= 16#d4e5;
    GB2312[4986]:= 16#debd;
    GB2312[4987]:= 16#debf;
    GB2312[4988]:= 16#c4a2;
    GB2312[4989]:= 16#dec1;
    GB2312[4990]:= 16#debe;
    GB2312[4991]:= 16#dec0;
    GB2312[4992]:= 16#d5ba;
    GB2312[4993]:= 16#dec2;
    GB2312[4994]:= 16#f2ae;
    GB2312[4995]:= 16#bba2;
    GB2312[4996]:= 16#c2b2;
    GB2312[4997]:= 16#c5b0;
    GB2312[4998]:= 16#c2c7;
    GB2312[4999]:= 16#f2af;          //GB2312码 4000-4999
END_IF;
(* Rung 16 *)
IF P_On THEN
    GB2312[5000]:= 16#d0e9;
    GB2312[5001]:= 16#d3dd;
    GB2312[5002]:= 16#ebbd;
    GB2312[5003]:= 16#b3e6;
    GB2312[5004]:= 16#f2b0;
    GB2312[5005]:= 16#f2b1;
    GB2312[5006]:= 16#caad;
    GB2312[5007]:= 16#bae7;
    GB2312[5008]:= 16#f2b3;
    GB2312[5009]:= 16#f2b5;
    GB2312[5010]:= 16#f2b4;
    GB2312[5011]:= 16#cbe4;
    GB2312[5012]:= 16#cfba;
    GB2312[5013]:= 16#f2b2;
    GB2312[5014]:= 16#cab4;
    GB2312[5015]:= 16#d2cf;
    GB2312[5016]:= 16#c2ec;
    GB2312[5017]:= 16#cec3;
    GB2312[5018]:= 16#f2b8;
    GB2312[5019]:= 16#b0f6;
    GB2312[5020]:= 16#f2b7;
    GB2312[5021]:= 16#f2be;
    GB2312[5022]:= 16#b2cf;
    GB2312[5023]:= 16#d1c1;
    GB2312[5024]:= 16#f2ba;
    GB2312[5025]:= 16#f2bc;
    GB2312[5026]:= 16#d4e9;
    GB2312[5027]:= 16#f2bb;
    GB2312[5028]:= 16#f2b6;
    GB2312[5029]:= 16#f2bf;
    GB2312[5030]:= 16#f2bd;
    GB2312[5031]:= 16#f2b9;
    GB2312[5032]:= 16#f2c7;
    GB2312[5033]:= 16#f2c4;
    GB2312[5034]:= 16#f2c6;
    GB2312[5035]:= 16#f2ca;
    GB2312[5036]:= 16#f2c2;
    GB2312[5037]:= 16#f2c0;
    GB2312[5038]:= 16#f2c5;
    GB2312[5039]:= 16#d6fb;
    GB2312[5040]:= 16#f2c1;
    GB2312[5041]:= 16#c7f9;
    GB2312[5042]:= 16#c9df;
    GB2312[5043]:= 16#f2c8;
    GB2312[5044]:= 16#b9c6;
    GB2312[5045]:= 16#b5b0;
    GB2312[5046]:= 16#f2c3;
    GB2312[5047]:= 16#f2c9;
    GB2312[5048]:= 16#f2d0;
    GB2312[5049]:= 16#f2d6;
    GB2312[5050]:= 16#bbd7;
    GB2312[5051]:= 16#f2d5;
    GB2312[5052]:= 16#cddc;
    GB2312[5053]:= 16#d6eb;
    GB2312[5054]:= 16#f2d2;
    GB2312[5055]:= 16#f2d4;
    GB2312[5056]:= 16#b8f2;
    GB2312[5057]:= 16#f2cb;
    GB2312[5058]:= 16#f2ce;
    GB2312[5059]:= 16#c2f9;
    GB2312[5060]:= 16#d5dd;
    GB2312[5061]:= 16#f2cc;
    GB2312[5062]:= 16#f2cd;
    GB2312[5063]:= 16#f2cf;
    GB2312[5064]:= 16#f2d3;
    GB2312[5065]:= 16#f2d9;
    GB2312[5066]:= 16#d3bc;
    GB2312[5067]:= 16#b6ea;
    GB2312[5068]:= 16#caf1;
    GB2312[5069]:= 16#b7e4;
    GB2312[5070]:= 16#f2d7;
    GB2312[5071]:= 16#f2d8;
    GB2312[5072]:= 16#f2da;
    GB2312[5073]:= 16#f2dd;
    GB2312[5074]:= 16#f2db;
    GB2312[5075]:= 16#f2dc;
    GB2312[5076]:= 16#d1d1;
    GB2312[5077]:= 16#f2d1;
    GB2312[5078]:= 16#cdc9;
    GB2312[5079]:= 16#cecf;
    GB2312[5080]:= 16#d6a9;
    GB2312[5081]:= 16#f2e3;
    GB2312[5082]:= 16#c3db;
    GB2312[5083]:= 16#f2e0;
    GB2312[5084]:= 16#c0af;
    GB2312[5085]:= 16#f2ec;
    GB2312[5086]:= 16#f2de;
    GB2312[5087]:= 16#f2e1;
    GB2312[5088]:= 16#f2e8;
    GB2312[5089]:= 16#f2e2;
    GB2312[5090]:= 16#f2e7;
    GB2312[5091]:= 16#f2e6;
    GB2312[5092]:= 16#f2e9;
    GB2312[5093]:= 16#f2df;
    GB2312[5094]:= 16#f2e4;
    GB2312[5095]:= 16#f2ea;
    GB2312[5096]:= 16#d3ac;
    GB2312[5097]:= 16#f2e5;
    GB2312[5098]:= 16#b2f5;
    GB2312[5099]:= 16#f2f2;
    GB2312[5100]:= 16#d0ab;
    GB2312[5101]:= 16#f2f5;
    GB2312[5102]:= 16#bbc8;
    GB2312[5103]:= 16#f2f9;
    GB2312[5104]:= 16#f2f0;
    GB2312[5105]:= 16#f2f6;
    GB2312[5106]:= 16#f2f8;
    GB2312[5107]:= 16#f2fa;
    GB2312[5108]:= 16#f2f3;
    GB2312[5109]:= 16#f2f1;
    GB2312[5110]:= 16#bafb;
    GB2312[5111]:= 16#b5fb;
    GB2312[5112]:= 16#f2ef;
    GB2312[5113]:= 16#f2f7;
    GB2312[5114]:= 16#f2ed;
    GB2312[5115]:= 16#f2ee;
    GB2312[5116]:= 16#f2eb;
    GB2312[5117]:= 16#f3a6;
    GB2312[5118]:= 16#f3a3;
    GB2312[5119]:= 16#f3a2;
    GB2312[5120]:= 16#f2f4;
    GB2312[5121]:= 16#c8da;
    GB2312[5122]:= 16#f2fb;
    GB2312[5123]:= 16#f3a5;
    GB2312[5124]:= 16#c3f8;
    GB2312[5125]:= 16#f2fd;
    GB2312[5126]:= 16#f3a7;
    GB2312[5127]:= 16#f3a9;
    GB2312[5128]:= 16#f3a4;
    GB2312[5129]:= 16#f2fc;
    GB2312[5130]:= 16#f3ab;
    GB2312[5131]:= 16#f3aa;
    GB2312[5132]:= 16#c2dd;
    GB2312[5133]:= 16#f3ae;
    GB2312[5134]:= 16#f3b0;
    GB2312[5135]:= 16#f3a1;
    GB2312[5136]:= 16#f3b1;
    GB2312[5137]:= 16#f3ac;
    GB2312[5138]:= 16#f3af;
    GB2312[5139]:= 16#f2fe;
    GB2312[5140]:= 16#f3ad;
    GB2312[5141]:= 16#f3b2;
    GB2312[5142]:= 16#f3b4;
    GB2312[5143]:= 16#f3a8;
    GB2312[5144]:= 16#f3b3;
    GB2312[5145]:= 16#f3b5;
    GB2312[5146]:= 16#d0b7;
    GB2312[5147]:= 16#f3b8;
    GB2312[5148]:= 16#d9f9;
    GB2312[5149]:= 16#f3b9;
    GB2312[5150]:= 16#f3b7;
    GB2312[5151]:= 16#c8e4;
    GB2312[5152]:= 16#f3b6;
    GB2312[5153]:= 16#f3ba;
    GB2312[5154]:= 16#f3bb;
    GB2312[5155]:= 16#b4c0;
    GB2312[5156]:= 16#eec3;
    GB2312[5157]:= 16#f3bc;
    GB2312[5158]:= 16#f3bd;
    GB2312[5159]:= 16#d1aa;
    GB2312[5160]:= 16#f4ac;
    GB2312[5161]:= 16#d0c6;
    GB2312[5162]:= 16#d0d0;
    GB2312[5163]:= 16#d1dc;
    GB2312[5164]:= 16#cfce;
    GB2312[5165]:= 16#bdd6;
    GB2312[5166]:= 16#d1c3;
    GB2312[5167]:= 16#bae2;
    GB2312[5168]:= 16#e1e9;
    GB2312[5169]:= 16#d2c2;
    GB2312[5170]:= 16#f1c2;
    GB2312[5171]:= 16#b2b9;
    GB2312[5172]:= 16#b1ed;
    GB2312[5173]:= 16#f1c3;
    GB2312[5174]:= 16#c9c0;
    GB2312[5175]:= 16#b3c4;
    GB2312[5176]:= 16#d9f2;
    GB2312[5177]:= 16#cba5;
    GB2312[5178]:= 16#f1c4;
    GB2312[5179]:= 16#d6d4;
    GB2312[5180]:= 16#f1c5;
    GB2312[5181]:= 16#f4c0;
    GB2312[5182]:= 16#f1c6;
    GB2312[5183]:= 16#d4ac;
    GB2312[5184]:= 16#f1c7;
    GB2312[5185]:= 16#b0c0;
    GB2312[5186]:= 16#f4c1;
    GB2312[5187]:= 16#f4c2;
    GB2312[5188]:= 16#b4fc;
    GB2312[5189]:= 16#c5db;
    GB2312[5190]:= 16#ccbb;
    GB2312[5191]:= 16#d0e4;
    GB2312[5192]:= 16#cde0;
    GB2312[5193]:= 16#f1c8;
    GB2312[5194]:= 16#d9f3;
    GB2312[5195]:= 16#b1bb;
    GB2312[5196]:= 16#cfae;
    GB2312[5197]:= 16#b8a4;
    GB2312[5198]:= 16#f1ca;
    GB2312[5199]:= 16#f1cb;
    GB2312[5200]:= 16#b2c3;
    GB2312[5201]:= 16#c1d1;
    GB2312[5202]:= 16#d7b0;
    GB2312[5203]:= 16#f1c9;
    GB2312[5204]:= 16#f1cc;
    GB2312[5205]:= 16#f1ce;
    GB2312[5206]:= 16#d9f6;
    GB2312[5207]:= 16#d2e1;
    GB2312[5208]:= 16#d4a3;
    GB2312[5209]:= 16#f4c3;
    GB2312[5210]:= 16#c8b9;
    GB2312[5211]:= 16#f4c4;
    GB2312[5212]:= 16#f1cd;
    GB2312[5213]:= 16#f1cf;
    GB2312[5214]:= 16#bfe3;
    GB2312[5215]:= 16#f1d0;
    GB2312[5216]:= 16#f1d4;
    GB2312[5217]:= 16#f1d6;
    GB2312[5218]:= 16#f1d1;
    GB2312[5219]:= 16#c9d1;
    GB2312[5220]:= 16#c5e1;
    GB2312[5221]:= 16#c2e3;
    GB2312[5222]:= 16#b9fc;
    GB2312[5223]:= 16#f1d3;
    GB2312[5224]:= 16#f1d5;
    GB2312[5225]:= 16#b9d3;
    GB2312[5226]:= 16#f1db;
    GB2312[5227]:= 16#bad6;
    GB2312[5228]:= 16#b0fd;
    GB2312[5229]:= 16#f1d9;
    GB2312[5230]:= 16#f1d8;
    GB2312[5231]:= 16#f1d2;
    GB2312[5232]:= 16#f1da;
    GB2312[5233]:= 16#f1d7;
    GB2312[5234]:= 16#c8ec;
    GB2312[5235]:= 16#cdca;
    GB2312[5236]:= 16#f1dd;
    GB2312[5237]:= 16#e5bd;
    GB2312[5238]:= 16#f1dc;
    GB2312[5239]:= 16#f1de;
    GB2312[5240]:= 16#f1df;
    GB2312[5241]:= 16#cfe5;
    GB2312[5242]:= 16#f4c5;
    GB2312[5243]:= 16#bdf3;
    GB2312[5244]:= 16#f1e0;
    GB2312[5245]:= 16#f1e1;
    GB2312[5246]:= 16#cef7;
    GB2312[5247]:= 16#d2aa;
    GB2312[5248]:= 16#f1fb;
    GB2312[5249]:= 16#b8b2;
    GB2312[5250]:= 16#bcfb;
    GB2312[5251]:= 16#b9db;
    GB2312[5252]:= 16#b9e6;
    GB2312[5253]:= 16#c3d9;
    GB2312[5254]:= 16#cad3;
    GB2312[5255]:= 16#eae8;
    GB2312[5256]:= 16#c0c0;
    GB2312[5257]:= 16#bef5;
    GB2312[5258]:= 16#eae9;
    GB2312[5259]:= 16#eaea;
    GB2312[5260]:= 16#eaeb;
    GB2312[5261]:= 16#eaec;
    GB2312[5262]:= 16#eaed;
    GB2312[5263]:= 16#eaee;
    GB2312[5264]:= 16#eaef;
    GB2312[5265]:= 16#bdc7;
    GB2312[5266]:= 16#f5fb;
    GB2312[5267]:= 16#f5fd;
    GB2312[5268]:= 16#f5fe;
    GB2312[5269]:= 16#f5fc;
    GB2312[5270]:= 16#bde2;
    GB2312[5271]:= 16#f6a1;
    GB2312[5272]:= 16#b4a5;
    GB2312[5273]:= 16#f6a2;
    GB2312[5274]:= 16#f6a3;
    GB2312[5275]:= 16#ecb2;
    GB2312[5276]:= 16#d1d4;
    GB2312[5277]:= 16#d9ea;
    GB2312[5278]:= 16#f6a4;
    GB2312[5279]:= 16#eeba;
    GB2312[5280]:= 16#d5b2;
    GB2312[5281]:= 16#d3fe;
    GB2312[5282]:= 16#ccdc;
    GB2312[5283]:= 16#cac4;
    GB2312[5284]:= 16#e5c0;
    GB2312[5285]:= 16#f6a5;
    GB2312[5286]:= 16#beaf;
    GB2312[5287]:= 16#c6a9;
    GB2312[5288]:= 16#daa5;
    GB2312[5289]:= 16#bcc6;
    GB2312[5290]:= 16#b6a9;
    GB2312[5291]:= 16#b8bc;
    GB2312[5292]:= 16#c8cf;
    GB2312[5293]:= 16#bca5;
    GB2312[5294]:= 16#daa6;
    GB2312[5295]:= 16#daa7;
    GB2312[5296]:= 16#ccd6;
    GB2312[5297]:= 16#c8c3;
    GB2312[5298]:= 16#daa8;
    GB2312[5299]:= 16#c6fd;
    GB2312[5300]:= 16#d1b5;
    GB2312[5301]:= 16#d2e9;
    GB2312[5302]:= 16#d1b6;
    GB2312[5303]:= 16#bcc7;
    GB2312[5304]:= 16#bdb2;
    GB2312[5305]:= 16#bbe4;
    GB2312[5306]:= 16#daa9;
    GB2312[5307]:= 16#daaa;
    GB2312[5308]:= 16#d1c8;
    GB2312[5309]:= 16#daab;
    GB2312[5310]:= 16#d0ed;
    GB2312[5311]:= 16#b6ef;
    GB2312[5312]:= 16#c2db;
    GB2312[5313]:= 16#cbcf;
    GB2312[5314]:= 16#b7ed;
    GB2312[5315]:= 16#c9e8;
    GB2312[5316]:= 16#b7c3;
    GB2312[5317]:= 16#bef7;
    GB2312[5318]:= 16#d6a4;
    GB2312[5319]:= 16#daac;
    GB2312[5320]:= 16#daad;
    GB2312[5321]:= 16#c6c0;
    GB2312[5322]:= 16#d7e7;
    GB2312[5323]:= 16#cab6;
    GB2312[5324]:= 16#d5a9;
    GB2312[5325]:= 16#cbdf;
    GB2312[5326]:= 16#d5ef;
    GB2312[5327]:= 16#daae;
    GB2312[5328]:= 16#d6df;
    GB2312[5329]:= 16#b4ca;
    GB2312[5330]:= 16#dab0;
    GB2312[5331]:= 16#daaf;
    GB2312[5332]:= 16#d2eb;
    GB2312[5333]:= 16#dab1;
    GB2312[5334]:= 16#dab2;
    GB2312[5335]:= 16#dab3;
    GB2312[5336]:= 16#cad4;
    GB2312[5337]:= 16#dab4;
    GB2312[5338]:= 16#caab;
    GB2312[5339]:= 16#dab5;
    GB2312[5340]:= 16#dab6;
    GB2312[5341]:= 16#b3cf;
    GB2312[5342]:= 16#d6ef;
    GB2312[5343]:= 16#dab7;
    GB2312[5344]:= 16#bbb0;
    GB2312[5345]:= 16#b5ae;
    GB2312[5346]:= 16#dab8;
    GB2312[5347]:= 16#dab9;
    GB2312[5348]:= 16#b9ee;
    GB2312[5349]:= 16#d1af;
    GB2312[5350]:= 16#d2e8;
    GB2312[5351]:= 16#daba;
    GB2312[5352]:= 16#b8c3;
    GB2312[5353]:= 16#cfea;
    GB2312[5354]:= 16#b2ef;
    GB2312[5355]:= 16#dabb;
    GB2312[5356]:= 16#dabc;
    GB2312[5357]:= 16#bdeb;
    GB2312[5358]:= 16#cedc;
    GB2312[5359]:= 16#d3ef;
    GB2312[5360]:= 16#dabd;
    GB2312[5361]:= 16#cef3;
    GB2312[5362]:= 16#dabe;
    GB2312[5363]:= 16#d3d5;
    GB2312[5364]:= 16#bbe5;
    GB2312[5365]:= 16#dabf;
    GB2312[5366]:= 16#cbb5;
    GB2312[5367]:= 16#cbd0;
    GB2312[5368]:= 16#dac0;
    GB2312[5369]:= 16#c7eb;
    GB2312[5370]:= 16#d6ee;
    GB2312[5371]:= 16#dac1;
    GB2312[5372]:= 16#c5b5;
    GB2312[5373]:= 16#b6c1;
    GB2312[5374]:= 16#dac2;
    GB2312[5375]:= 16#b7cc;
    GB2312[5376]:= 16#bfce;
    GB2312[5377]:= 16#dac3;
    GB2312[5378]:= 16#dac4;
    GB2312[5379]:= 16#cbad;
    GB2312[5380]:= 16#dac5;
    GB2312[5381]:= 16#b5f7;
    GB2312[5382]:= 16#dac6;
    GB2312[5383]:= 16#c1c2;
    GB2312[5384]:= 16#d7bb;
    GB2312[5385]:= 16#dac7;
    GB2312[5386]:= 16#ccb8;
    GB2312[5387]:= 16#d2ea;
    GB2312[5388]:= 16#c4b1;
    GB2312[5389]:= 16#dac8;
    GB2312[5390]:= 16#b5fd;
    GB2312[5391]:= 16#bbd1;
    GB2312[5392]:= 16#dac9;
    GB2312[5393]:= 16#d0b3;
    GB2312[5394]:= 16#daca;
    GB2312[5395]:= 16#dacb;
    GB2312[5396]:= 16#cebd;
    GB2312[5397]:= 16#dacc;
    GB2312[5398]:= 16#dacd;
    GB2312[5399]:= 16#dace;
    GB2312[5400]:= 16#b2f7;
    GB2312[5401]:= 16#dad1;
    GB2312[5402]:= 16#dacf;
    GB2312[5403]:= 16#d1e8;
    GB2312[5404]:= 16#dad0;
    GB2312[5405]:= 16#c3d5;
    GB2312[5406]:= 16#dad2;
    GB2312[5407]:= 16#dad3;
    GB2312[5408]:= 16#dad4;
    GB2312[5409]:= 16#dad5;
    GB2312[5410]:= 16#d0bb;
    GB2312[5411]:= 16#d2a5;
    GB2312[5412]:= 16#b0f9;
    GB2312[5413]:= 16#dad6;
    GB2312[5414]:= 16#c7ab;
    GB2312[5415]:= 16#dad7;
    GB2312[5416]:= 16#bdf7;
    GB2312[5417]:= 16#c3a1;
    GB2312[5418]:= 16#dad8;
    GB2312[5419]:= 16#dad9;
    GB2312[5420]:= 16#c3fd;
    GB2312[5421]:= 16#ccb7;
    GB2312[5422]:= 16#dada;
    GB2312[5423]:= 16#dadb;
    GB2312[5424]:= 16#c0be;
    GB2312[5425]:= 16#c6d7;
    GB2312[5426]:= 16#dadc;
    GB2312[5427]:= 16#dadd;
    GB2312[5428]:= 16#c7b4;
    GB2312[5429]:= 16#dade;
    GB2312[5430]:= 16#dadf;
    GB2312[5431]:= 16#b9c8;
    GB2312[5432]:= 16#bbed;
    GB2312[5433]:= 16#b6b9;
    GB2312[5434]:= 16#f4f8;
    GB2312[5435]:= 16#f4f9;
    GB2312[5436]:= 16#cde3;
    GB2312[5437]:= 16#f5b9;
    GB2312[5438]:= 16#ebe0;
    GB2312[5439]:= 16#cff3;
    GB2312[5440]:= 16#bbbf;
    GB2312[5441]:= 16#bac0;
    GB2312[5442]:= 16#d4a5;
    GB2312[5443]:= 16#e1d9;
    GB2312[5444]:= 16#f5f4;
    GB2312[5445]:= 16#b1aa;
    GB2312[5446]:= 16#b2f2;
    GB2312[5447]:= 16#f5f5;
    GB2312[5448]:= 16#f5f7;
    GB2312[5449]:= 16#bad1;
    GB2312[5450]:= 16#f5f6;
    GB2312[5451]:= 16#c3b2;
    GB2312[5452]:= 16#f5f9;
    GB2312[5453]:= 16#f5f8;
    GB2312[5454]:= 16#b1b4;
    GB2312[5455]:= 16#d5ea;
    GB2312[5456]:= 16#b8ba;
    GB2312[5457]:= 16#b9b1;
    GB2312[5458]:= 16#b2c6;
    GB2312[5459]:= 16#d4f0;
    GB2312[5460]:= 16#cfcd;
    GB2312[5461]:= 16#b0dc;
    GB2312[5462]:= 16#d5cb;
    GB2312[5463]:= 16#bbf5;
    GB2312[5464]:= 16#d6ca;
    GB2312[5465]:= 16#b7b7;
    GB2312[5466]:= 16#ccb0;
    GB2312[5467]:= 16#c6b6;
    GB2312[5468]:= 16#b1e1;
    GB2312[5469]:= 16#b9ba;
    GB2312[5470]:= 16#d6fc;
    GB2312[5471]:= 16#b9e1;
    GB2312[5472]:= 16#b7a1;
    GB2312[5473]:= 16#bcfa;
    GB2312[5474]:= 16#eada;
    GB2312[5475]:= 16#eadb;
    GB2312[5476]:= 16#ccf9;
    GB2312[5477]:= 16#b9f3;
    GB2312[5478]:= 16#eadc;
    GB2312[5479]:= 16#b4fb;
    GB2312[5480]:= 16#c3b3;
    GB2312[5481]:= 16#b7d1;
    GB2312[5482]:= 16#bad8;
    GB2312[5483]:= 16#eadd;
    GB2312[5484]:= 16#d4f4;
    GB2312[5485]:= 16#eade;
    GB2312[5486]:= 16#bcd6;
    GB2312[5487]:= 16#bbdf;
    GB2312[5488]:= 16#eadf;
    GB2312[5489]:= 16#c1de;
    GB2312[5490]:= 16#c2b8;
    GB2312[5491]:= 16#d4df;
    GB2312[5492]:= 16#d7ca;
    GB2312[5493]:= 16#eae0;
    GB2312[5494]:= 16#eae1;
    GB2312[5495]:= 16#eae4;
    GB2312[5496]:= 16#eae2;
    GB2312[5497]:= 16#eae3;
    GB2312[5498]:= 16#c9de;
    GB2312[5499]:= 16#b8b3;
    GB2312[5500]:= 16#b6c4;
    GB2312[5501]:= 16#eae5;
    GB2312[5502]:= 16#caea;
    GB2312[5503]:= 16#c9cd;
    GB2312[5504]:= 16#b4cd;
    GB2312[5505]:= 16#e2d9;
    GB2312[5506]:= 16#c5e2;
    GB2312[5507]:= 16#eae6;
    GB2312[5508]:= 16#c0b5;
    GB2312[5509]:= 16#d7b8;
    GB2312[5510]:= 16#eae7;
    GB2312[5511]:= 16#d7ac;
    GB2312[5512]:= 16#c8fc;
    GB2312[5513]:= 16#d8d3;
    GB2312[5514]:= 16#d8cd;
    GB2312[5515]:= 16#d4de;
    GB2312[5516]:= 16#d4f9;
    GB2312[5517]:= 16#c9c4;
    GB2312[5518]:= 16#d3ae;
    GB2312[5519]:= 16#b8d3;
    GB2312[5520]:= 16#b3e0;
    GB2312[5521]:= 16#c9e2;
    GB2312[5522]:= 16#f4f6;
    GB2312[5523]:= 16#bad5;
    GB2312[5524]:= 16#f4f7;
    GB2312[5525]:= 16#d7df;
    GB2312[5526]:= 16#f4f1;
    GB2312[5527]:= 16#b8b0;
    GB2312[5528]:= 16#d5d4;
    GB2312[5529]:= 16#b8cf;
    GB2312[5530]:= 16#c6f0;
    GB2312[5531]:= 16#b3c3;
    GB2312[5532]:= 16#f4f2;
    GB2312[5533]:= 16#b3ac;
    GB2312[5534]:= 16#d4bd;
    GB2312[5535]:= 16#c7f7;
    GB2312[5536]:= 16#f4f4;
    GB2312[5537]:= 16#f4f3;
    GB2312[5538]:= 16#cccb;
    GB2312[5539]:= 16#c8a4;
    GB2312[5540]:= 16#f4f5;
    GB2312[5541]:= 16#d7e3;
    GB2312[5542]:= 16#c5bf;
    GB2312[5543]:= 16#f5c0;
    GB2312[5544]:= 16#f5bb;
    GB2312[5545]:= 16#f5c3;
    GB2312[5546]:= 16#f5c2;
    GB2312[5547]:= 16#d6ba;
    GB2312[5548]:= 16#f5c1;
    GB2312[5549]:= 16#d4be;
    GB2312[5550]:= 16#f5c4;
    GB2312[5551]:= 16#f5cc;
    GB2312[5552]:= 16#b0cf;
    GB2312[5553]:= 16#b5f8;
    GB2312[5554]:= 16#f5c9;
    GB2312[5555]:= 16#f5ca;
    GB2312[5556]:= 16#c5dc;
    GB2312[5557]:= 16#f5c5;
    GB2312[5558]:= 16#f5c6;
    GB2312[5559]:= 16#f5c7;
    GB2312[5560]:= 16#f5cb;
    GB2312[5561]:= 16#bee0;
    GB2312[5562]:= 16#f5c8;
    GB2312[5563]:= 16#b8fa;
    GB2312[5564]:= 16#f5d0;
    GB2312[5565]:= 16#f5d3;
    GB2312[5566]:= 16#bfe7;
    GB2312[5567]:= 16#b9f2;
    GB2312[5568]:= 16#f5bc;
    GB2312[5569]:= 16#f5cd;
    GB2312[5570]:= 16#c2b7;
    GB2312[5571]:= 16#ccf8;
    GB2312[5572]:= 16#bcf9;
    GB2312[5573]:= 16#f5ce;
    GB2312[5574]:= 16#f5cf;
    GB2312[5575]:= 16#f5d1;
    GB2312[5576]:= 16#b6e5;
    GB2312[5577]:= 16#f5d2;
    GB2312[5578]:= 16#f5d5;
    GB2312[5579]:= 16#f5bd;
    GB2312[5580]:= 16#f5d4;
    GB2312[5581]:= 16#d3bb;
    GB2312[5582]:= 16#b3ec;
    GB2312[5583]:= 16#cca4;
    GB2312[5584]:= 16#f5d6;
    GB2312[5585]:= 16#f5d7;
    GB2312[5586]:= 16#bee1;
    GB2312[5587]:= 16#f5d8;
    GB2312[5588]:= 16#ccdf;
    GB2312[5589]:= 16#f5db;
    GB2312[5590]:= 16#b2c8;
    GB2312[5591]:= 16#d7d9;
    GB2312[5592]:= 16#f5d9;
    GB2312[5593]:= 16#f5da;
    GB2312[5594]:= 16#f5dc;
    GB2312[5595]:= 16#f5e2;
    GB2312[5596]:= 16#f5e0;
    GB2312[5597]:= 16#f5df;
    GB2312[5598]:= 16#f5dd;
    GB2312[5599]:= 16#f5e1;
    GB2312[5600]:= 16#f5de;
    GB2312[5601]:= 16#f5e4;
    GB2312[5602]:= 16#f5e5;
    GB2312[5603]:= 16#cce3;
    GB2312[5604]:= 16#e5bf;
    GB2312[5605]:= 16#b5b8;
    GB2312[5606]:= 16#f5e3;
    GB2312[5607]:= 16#f5e8;
    GB2312[5608]:= 16#cca3;
    GB2312[5609]:= 16#f5e6;
    GB2312[5610]:= 16#f5e7;
    GB2312[5611]:= 16#f5be;
    GB2312[5612]:= 16#b1c4;
    GB2312[5613]:= 16#f5bf;
    GB2312[5614]:= 16#b5c5;
    GB2312[5615]:= 16#b2e4;
    GB2312[5616]:= 16#f5ec;
    GB2312[5617]:= 16#f5e9;
    GB2312[5618]:= 16#b6d7;
    GB2312[5619]:= 16#f5ed;
    GB2312[5620]:= 16#f5ea;
    GB2312[5621]:= 16#f5eb;
    GB2312[5622]:= 16#b4da;
    GB2312[5623]:= 16#d4ea;
    GB2312[5624]:= 16#f5ee;
    GB2312[5625]:= 16#b3f9;
    GB2312[5626]:= 16#f5ef;
    GB2312[5627]:= 16#f5f1;
    GB2312[5628]:= 16#f5f0;
    GB2312[5629]:= 16#f5f2;
    GB2312[5630]:= 16#f5f3;
    GB2312[5631]:= 16#c9ed;
    GB2312[5632]:= 16#b9aa;
    GB2312[5633]:= 16#c7fb;
    GB2312[5634]:= 16#b6e3;
    GB2312[5635]:= 16#ccc9;
    GB2312[5636]:= 16#eaa6;
    GB2312[5637]:= 16#b3b5;
    GB2312[5638]:= 16#d4fe;
    GB2312[5639]:= 16#b9ec;
    GB2312[5640]:= 16#d0f9;
    GB2312[5641]:= 16#e9ed;
    GB2312[5642]:= 16#d7aa;
    GB2312[5643]:= 16#e9ee;
    GB2312[5644]:= 16#c2d6;
    GB2312[5645]:= 16#c8ed;
    GB2312[5646]:= 16#bae4;
    GB2312[5647]:= 16#e9ef;
    GB2312[5648]:= 16#e9f0;
    GB2312[5649]:= 16#e9f1;
    GB2312[5650]:= 16#d6e1;
    GB2312[5651]:= 16#e9f2;
    GB2312[5652]:= 16#e9f3;
    GB2312[5653]:= 16#e9f5;
    GB2312[5654]:= 16#e9f4;
    GB2312[5655]:= 16#e9f6;
    GB2312[5656]:= 16#e9f7;
    GB2312[5657]:= 16#c7e1;
    GB2312[5658]:= 16#e9f8;
    GB2312[5659]:= 16#d4d8;
    GB2312[5660]:= 16#e9f9;
    GB2312[5661]:= 16#bdce;
    GB2312[5662]:= 16#e9fa;
    GB2312[5663]:= 16#e9fb;
    GB2312[5664]:= 16#bdcf;
    GB2312[5665]:= 16#e9fc;
    GB2312[5666]:= 16#b8a8;
    GB2312[5667]:= 16#c1be;
    GB2312[5668]:= 16#e9fd;
    GB2312[5669]:= 16#b1b2;
    GB2312[5670]:= 16#bbd4;
    GB2312[5671]:= 16#b9f5;
    GB2312[5672]:= 16#e9fe;
    GB2312[5673]:= 16#eaa1;
    GB2312[5674]:= 16#eaa2;
    GB2312[5675]:= 16#eaa3;
    GB2312[5676]:= 16#b7f8;
    GB2312[5677]:= 16#bcad;
    GB2312[5678]:= 16#cae4;
    GB2312[5679]:= 16#e0ce;
    GB2312[5680]:= 16#d4af;
    GB2312[5681]:= 16#cfbd;
    GB2312[5682]:= 16#d5b7;
    GB2312[5683]:= 16#eaa4;
    GB2312[5684]:= 16#d5de;
    GB2312[5685]:= 16#eaa5;
    GB2312[5686]:= 16#d0c1;
    GB2312[5687]:= 16#b9bc;
    GB2312[5688]:= 16#b4c7;
    GB2312[5689]:= 16#b1d9;
    GB2312[5690]:= 16#c0b1;
    GB2312[5691]:= 16#b1e6;
    GB2312[5692]:= 16#b1e7;
    GB2312[5693]:= 16#b1e8;
    GB2312[5694]:= 16#b3bd;
    GB2312[5695]:= 16#c8e8;
    GB2312[5696]:= 16#e5c1;
    GB2312[5697]:= 16#b1df;
    GB2312[5698]:= 16#c1c9;
    GB2312[5699]:= 16#b4ef;
    GB2312[5700]:= 16#c7a8;
    GB2312[5701]:= 16#d3d8;
    GB2312[5702]:= 16#c6f9;
    GB2312[5703]:= 16#d1b8;
    GB2312[5704]:= 16#b9fd;
    GB2312[5705]:= 16#c2f5;
    GB2312[5706]:= 16#d3ad;
    GB2312[5707]:= 16#d4cb;
    GB2312[5708]:= 16#bdfc;
    GB2312[5709]:= 16#e5c2;
    GB2312[5710]:= 16#b7b5;
    GB2312[5711]:= 16#e5c3;
    GB2312[5712]:= 16#bbb9;
    GB2312[5713]:= 16#d5e2;
    GB2312[5714]:= 16#bdf8;
    GB2312[5715]:= 16#d4b6;
    GB2312[5716]:= 16#cea5;
    GB2312[5717]:= 16#c1ac;
    GB2312[5718]:= 16#b3d9;
    GB2312[5719]:= 16#ccf6;
    GB2312[5720]:= 16#e5c6;
    GB2312[5721]:= 16#e5c4;
    GB2312[5722]:= 16#e5c8;
    GB2312[5723]:= 16#e5ca;
    GB2312[5724]:= 16#e5c7;
    GB2312[5725]:= 16#b5cf;
    GB2312[5726]:= 16#c6c8;
    GB2312[5727]:= 16#b5fc;
    GB2312[5728]:= 16#e5c5;
    GB2312[5729]:= 16#caf6;
    GB2312[5730]:= 16#e5c9;
    GB2312[5731]:= 16#c3d4;
    GB2312[5732]:= 16#b1c5;
    GB2312[5733]:= 16#bca3;
    GB2312[5734]:= 16#d7b7;
    GB2312[5735]:= 16#cdcb;
    GB2312[5736]:= 16#cbcd;
    GB2312[5737]:= 16#caca;
    GB2312[5738]:= 16#ccd3;
    GB2312[5739]:= 16#e5cc;
    GB2312[5740]:= 16#e5cb;
    GB2312[5741]:= 16#c4e6;
    GB2312[5742]:= 16#d1a1;
    GB2312[5743]:= 16#d1b7;
    GB2312[5744]:= 16#e5cd;
    GB2312[5745]:= 16#e5d0;
    GB2312[5746]:= 16#cdb8;
    GB2312[5747]:= 16#d6f0;
    GB2312[5748]:= 16#e5cf;
    GB2312[5749]:= 16#b5dd;
    GB2312[5750]:= 16#cdbe;
    GB2312[5751]:= 16#e5d1;
    GB2312[5752]:= 16#b6ba;
    GB2312[5753]:= 16#cda8;
    GB2312[5754]:= 16#b9e4;
    GB2312[5755]:= 16#cac5;
    GB2312[5756]:= 16#b3d1;
    GB2312[5757]:= 16#cbd9;
    GB2312[5758]:= 16#d4ec;
    GB2312[5759]:= 16#e5d2;
    GB2312[5760]:= 16#b7ea;
    GB2312[5761]:= 16#e5ce;
    GB2312[5762]:= 16#e5d5;
    GB2312[5763]:= 16#b4fe;
    GB2312[5764]:= 16#e5d6;
    GB2312[5765]:= 16#e5d3;
    GB2312[5766]:= 16#e5d4;
    GB2312[5767]:= 16#d2dd;
    GB2312[5768]:= 16#c2df;
    GB2312[5769]:= 16#b1c6;
    GB2312[5770]:= 16#d3e2;
    GB2312[5771]:= 16#b6dd;
    GB2312[5772]:= 16#cbec;
    GB2312[5773]:= 16#e5d7;
    GB2312[5774]:= 16#d3f6;
    GB2312[5775]:= 16#b1e9;
    GB2312[5776]:= 16#b6f4;
    GB2312[5777]:= 16#e5da;
    GB2312[5778]:= 16#e5d8;
    GB2312[5779]:= 16#e5d9;
    GB2312[5780]:= 16#b5c0;
    GB2312[5781]:= 16#d2c5;
    GB2312[5782]:= 16#e5dc;
    GB2312[5783]:= 16#e5de;
    GB2312[5784]:= 16#e5dd;
    GB2312[5785]:= 16#c7b2;
    GB2312[5786]:= 16#d2a3;
    GB2312[5787]:= 16#e5db;
    GB2312[5788]:= 16#d4e2;
    GB2312[5789]:= 16#d5da;
    GB2312[5790]:= 16#e5e0;
    GB2312[5791]:= 16#d7f1;
    GB2312[5792]:= 16#e5e1;
    GB2312[5793]:= 16#b1dc;
    GB2312[5794]:= 16#d1fb;
    GB2312[5795]:= 16#e5e2;
    GB2312[5796]:= 16#e5e4;
    GB2312[5797]:= 16#e5e3;
    GB2312[5798]:= 16#e5e5;
    GB2312[5799]:= 16#d2d8;
    GB2312[5800]:= 16#b5cb;
    GB2312[5801]:= 16#e7df;
    GB2312[5802]:= 16#daf5;
    GB2312[5803]:= 16#daf8;
    GB2312[5804]:= 16#daf6;
    GB2312[5805]:= 16#daf7;
    GB2312[5806]:= 16#dafa;
    GB2312[5807]:= 16#d0cf;
    GB2312[5808]:= 16#c4c7;
    GB2312[5809]:= 16#b0ee;
    GB2312[5810]:= 16#d0b0;
    GB2312[5811]:= 16#daf9;
    GB2312[5812]:= 16#d3ca;
    GB2312[5813]:= 16#baaa;
    GB2312[5814]:= 16#dba2;
    GB2312[5815]:= 16#c7f1;
    GB2312[5816]:= 16#dafc;
    GB2312[5817]:= 16#dafb;
    GB2312[5818]:= 16#c9db;
    GB2312[5819]:= 16#dafd;
    GB2312[5820]:= 16#dba1;
    GB2312[5821]:= 16#d7de;
    GB2312[5822]:= 16#dafe;
    GB2312[5823]:= 16#c1da;
    GB2312[5824]:= 16#dba5;
    GB2312[5825]:= 16#d3f4;
    GB2312[5826]:= 16#dba7;
    GB2312[5827]:= 16#dba4;
    GB2312[5828]:= 16#dba8;
    GB2312[5829]:= 16#bdbc;
    GB2312[5830]:= 16#c0c9;
    GB2312[5831]:= 16#dba3;
    GB2312[5832]:= 16#dba6;
    GB2312[5833]:= 16#d6a3;
    GB2312[5834]:= 16#dba9;
    GB2312[5835]:= 16#dbad;
    GB2312[5836]:= 16#dbae;
    GB2312[5837]:= 16#dbac;
    GB2312[5838]:= 16#bac2;
    GB2312[5839]:= 16#bfa4;
    GB2312[5840]:= 16#dbab;
    GB2312[5841]:= 16#dbaa;
    GB2312[5842]:= 16#d4c7;
    GB2312[5843]:= 16#b2bf;
    GB2312[5844]:= 16#dbaf;
    GB2312[5845]:= 16#b9f9;
    GB2312[5846]:= 16#dbb0;
    GB2312[5847]:= 16#b3bb;
    GB2312[5848]:= 16#b5a6;
    GB2312[5849]:= 16#b6bc;
    GB2312[5850]:= 16#dbb1;
    GB2312[5851]:= 16#b6f5;
    GB2312[5852]:= 16#dbb2;
    GB2312[5853]:= 16#b1c9;
    GB2312[5854]:= 16#dbb4;
    GB2312[5855]:= 16#dbb3;
    GB2312[5856]:= 16#dbb5;
    GB2312[5857]:= 16#dbb7;
    GB2312[5858]:= 16#dbb6;
    GB2312[5859]:= 16#dbb8;
    GB2312[5860]:= 16#dbb9;
    GB2312[5861]:= 16#dbba;
    GB2312[5862]:= 16#d3cf;
    GB2312[5863]:= 16#f4fa;
    GB2312[5864]:= 16#c7f5;
    GB2312[5865]:= 16#d7c3;
    GB2312[5866]:= 16#c5e4;
    GB2312[5867]:= 16#f4fc;
    GB2312[5868]:= 16#f4fd;
    GB2312[5869]:= 16#f4fb;
    GB2312[5870]:= 16#bec6;
    GB2312[5871]:= 16#d0ef;
    GB2312[5872]:= 16#b7d3;
    GB2312[5873]:= 16#d4cd;
    GB2312[5874]:= 16#ccaa;
    GB2312[5875]:= 16#f5a2;
    GB2312[5876]:= 16#f5a1;
    GB2312[5877]:= 16#baa8;
    GB2312[5878]:= 16#f4fe;
    GB2312[5879]:= 16#cbd6;
    GB2312[5880]:= 16#f5a4;
    GB2312[5881]:= 16#c0d2;
    GB2312[5882]:= 16#b3ea;
    GB2312[5883]:= 16#cdaa;
    GB2312[5884]:= 16#f5a5;
    GB2312[5885]:= 16#f5a3;
    GB2312[5886]:= 16#bdb4;
    GB2312[5887]:= 16#f5a8;
    GB2312[5888]:= 16#f5a9;
    GB2312[5889]:= 16#bdcd;
    GB2312[5890]:= 16#c3b8;
    GB2312[5891]:= 16#bfe1;
    GB2312[5892]:= 16#cbe1;
    GB2312[5893]:= 16#f5aa;
    GB2312[5894]:= 16#f5a6;
    GB2312[5895]:= 16#f5a7;
    GB2312[5896]:= 16#c4f0;
    GB2312[5897]:= 16#f5ac;
    GB2312[5898]:= 16#b4bc;
    GB2312[5899]:= 16#d7ed;
    GB2312[5900]:= 16#b4d7;
    GB2312[5901]:= 16#f5ab;
    GB2312[5902]:= 16#f5ae;
    GB2312[5903]:= 16#f5ad;
    GB2312[5904]:= 16#f5af;
    GB2312[5905]:= 16#d0d1;
    GB2312[5906]:= 16#c3d1;
    GB2312[5907]:= 16#c8a9;
    GB2312[5908]:= 16#f5b0;
    GB2312[5909]:= 16#f5b1;
    GB2312[5910]:= 16#f5b2;
    GB2312[5911]:= 16#f5b3;
    GB2312[5912]:= 16#f5b4;
    GB2312[5913]:= 16#f5b5;
    GB2312[5914]:= 16#f5b7;
    GB2312[5915]:= 16#f5b6;
    GB2312[5916]:= 16#f5b8;
    GB2312[5917]:= 16#b2c9;
    GB2312[5918]:= 16#d3d4;
    GB2312[5919]:= 16#cacd;
    GB2312[5920]:= 16#c0ef;
    GB2312[5921]:= 16#d6d8;
    GB2312[5922]:= 16#d2b0;
    GB2312[5923]:= 16#c1bf;
    GB2312[5924]:= 16#bdf0;
    GB2312[5925]:= 16#b8aa;
    GB2312[5926]:= 16#bcf8;
    GB2312[5927]:= 16#f6c6;
    GB2312[5928]:= 16#f6c7;
    GB2312[5929]:= 16#f6c8;
    GB2312[5930]:= 16#f6c9;
    GB2312[5931]:= 16#f6ca;
    GB2312[5932]:= 16#f6cc;
    GB2312[5933]:= 16#f6cb;
    GB2312[5934]:= 16#f7e9;
    GB2312[5935]:= 16#f6cd;
    GB2312[5936]:= 16#f6ce;
    GB2312[5937]:= 16#eec4;
    GB2312[5938]:= 16#eec5;
    GB2312[5939]:= 16#eec6;
    GB2312[5940]:= 16#d5eb;
    GB2312[5941]:= 16#b6a4;
    GB2312[5942]:= 16#eec8;
    GB2312[5943]:= 16#eec7;
    GB2312[5944]:= 16#eec9;
    GB2312[5945]:= 16#eeca;
    GB2312[5946]:= 16#c7a5;
    GB2312[5947]:= 16#eecb;
    GB2312[5948]:= 16#eecc;
    GB2312[5949]:= 16#b7b0;
    GB2312[5950]:= 16#b5f6;
    GB2312[5951]:= 16#eecd;
    GB2312[5952]:= 16#eecf;
    GB2312[5953]:= 16#eece;
    GB2312[5954]:= 16#b8c6;
    GB2312[5955]:= 16#eed0;
    GB2312[5956]:= 16#eed1;
    GB2312[5957]:= 16#eed2;
    GB2312[5958]:= 16#b6db;
    GB2312[5959]:= 16#b3ae;
    GB2312[5960]:= 16#d6d3;
    GB2312[5961]:= 16#c4c6;
    GB2312[5962]:= 16#b1b5;
    GB2312[5963]:= 16#b8d6;
    GB2312[5964]:= 16#eed3;
    GB2312[5965]:= 16#eed4;
    GB2312[5966]:= 16#d4bf;
    GB2312[5967]:= 16#c7d5;
    GB2312[5968]:= 16#befb;
    GB2312[5969]:= 16#ced9;
    GB2312[5970]:= 16#b9b3;
    GB2312[5971]:= 16#eed6;
    GB2312[5972]:= 16#eed5;
    GB2312[5973]:= 16#eed8;
    GB2312[5974]:= 16#eed7;
    GB2312[5975]:= 16#c5a5;
    GB2312[5976]:= 16#eed9;
    GB2312[5977]:= 16#eeda;
    GB2312[5978]:= 16#c7ae;
    GB2312[5979]:= 16#eedb;
    GB2312[5980]:= 16#c7af;
    GB2312[5981]:= 16#eedc;
    GB2312[5982]:= 16#b2a7;
    GB2312[5983]:= 16#eedd;
    GB2312[5984]:= 16#eede;
    GB2312[5985]:= 16#eedf;
    GB2312[5986]:= 16#eee0;
    GB2312[5987]:= 16#eee1;
    GB2312[5988]:= 16#d7ea;
    GB2312[5989]:= 16#eee2;
    GB2312[5990]:= 16#eee3;
    GB2312[5991]:= 16#bcd8;
    GB2312[5992]:= 16#eee4;
    GB2312[5993]:= 16#d3cb;
    GB2312[5994]:= 16#ccfa;
    GB2312[5995]:= 16#b2ac;
    GB2312[5996]:= 16#c1e5;
    GB2312[5997]:= 16#eee5;
    GB2312[5998]:= 16#c7a6;
    GB2312[5999]:= 16#c3ad;           //GB2312码 5000-5999
END_IF;

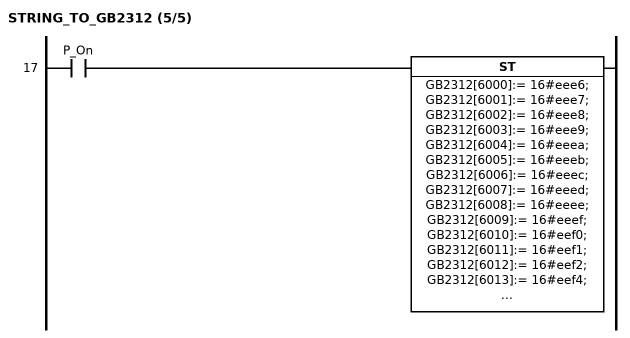
(* [picture p5: STRING_TO_GB2312, rungs 17-17] *)
(* Rung 17 *)
IF P_On THEN
    GB2312[6000]:= 16#eee6;
    GB2312[6001]:= 16#eee7;
    GB2312[6002]:= 16#eee8;
    GB2312[6003]:= 16#eee9;
    GB2312[6004]:= 16#eeea;
    GB2312[6005]:= 16#eeeb;
    GB2312[6006]:= 16#eeec;
    GB2312[6007]:= 16#eeed;
    GB2312[6008]:= 16#eeee;
    GB2312[6009]:= 16#eeef;
    GB2312[6010]:= 16#eef0;
    GB2312[6011]:= 16#eef1;
    GB2312[6012]:= 16#eef2;
    GB2312[6013]:= 16#eef4;
    GB2312[6014]:= 16#eef3;
    GB2312[6015]:= 16#eef5;
    GB2312[6016]:= 16#cdad;
    GB2312[6017]:= 16#c2c1;
    GB2312[6018]:= 16#eef6;
    GB2312[6019]:= 16#eef7;
    GB2312[6020]:= 16#eef8;
    GB2312[6021]:= 16#d5a1;
    GB2312[6022]:= 16#eef9;
    GB2312[6023]:= 16#cfb3;
    GB2312[6024]:= 16#eefa;
    GB2312[6025]:= 16#eefb;
    GB2312[6026]:= 16#eefc;
    GB2312[6027]:= 16#eefd;
    GB2312[6028]:= 16#efa1;
    GB2312[6029]:= 16#eefe;
    GB2312[6030]:= 16#efa2;
    GB2312[6031]:= 16#b8f5;
    GB2312[6032]:= 16#c3fa;
    GB2312[6033]:= 16#efa3;
    GB2312[6034]:= 16#efa4;
    GB2312[6035]:= 16#bdc2;
    GB2312[6036]:= 16#d2bf;
    GB2312[6037]:= 16#b2f9;
    GB2312[6038]:= 16#efa5;
    GB2312[6039]:= 16#efa6;
    GB2312[6040]:= 16#efa7;
    GB2312[6041]:= 16#d2f8;
    GB2312[6042]:= 16#efa8;
    GB2312[6043]:= 16#d6fd;
    GB2312[6044]:= 16#efa9;
    GB2312[6045]:= 16#c6cc;
    GB2312[6046]:= 16#efaa;
    GB2312[6047]:= 16#efab;
    GB2312[6048]:= 16#c1b4;
    GB2312[6049]:= 16#efac;
    GB2312[6050]:= 16#cffa;
    GB2312[6051]:= 16#cbf8;
    GB2312[6052]:= 16#efae;
    GB2312[6053]:= 16#efad;
    GB2312[6054]:= 16#b3fa;
    GB2312[6055]:= 16#b9f8;
    GB2312[6056]:= 16#efaf;
    GB2312[6057]:= 16#efb0;
    GB2312[6058]:= 16#d0e2;
    GB2312[6059]:= 16#efb1;
    GB2312[6060]:= 16#efb2;
    GB2312[6061]:= 16#b7e6;
    GB2312[6062]:= 16#d0bf;
    GB2312[6063]:= 16#efb3;
    GB2312[6064]:= 16#efb4;
    GB2312[6065]:= 16#efb5;
    GB2312[6066]:= 16#c8f1;
    GB2312[6067]:= 16#cce0;
    GB2312[6068]:= 16#efb6;
    GB2312[6069]:= 16#efb7;
    GB2312[6070]:= 16#efb8;
    GB2312[6071]:= 16#efb9;
    GB2312[6072]:= 16#efba;
    GB2312[6073]:= 16#d5e0;
    GB2312[6074]:= 16#efbb;
    GB2312[6075]:= 16#b4ed;
    GB2312[6076]:= 16#c3aa;
    GB2312[6077]:= 16#efbc;
    GB2312[6078]:= 16#efbd;
    GB2312[6079]:= 16#efbe;
    GB2312[6080]:= 16#efbf;
    GB2312[6081]:= 16#cefd;
    GB2312[6082]:= 16#efc0;
    GB2312[6083]:= 16#c2e0;
    GB2312[6084]:= 16#b4b8;
    GB2312[6085]:= 16#d7b6;
    GB2312[6086]:= 16#bdf5;
    GB2312[6087]:= 16#cfc7;
    GB2312[6088]:= 16#efc3;
    GB2312[6089]:= 16#efc1;
    GB2312[6090]:= 16#efc2;
    GB2312[6091]:= 16#efc4;
    GB2312[6092]:= 16#b6a7;
    GB2312[6093]:= 16#bcfc;
    GB2312[6094]:= 16#bee2;
    GB2312[6095]:= 16#c3cc;
    GB2312[6096]:= 16#efc5;
    GB2312[6097]:= 16#efc6;
    GB2312[6098]:= 16#efc7;
    GB2312[6099]:= 16#efcf;
    GB2312[6100]:= 16#efc8;
    GB2312[6101]:= 16#efc9;
    GB2312[6102]:= 16#efca;
    GB2312[6103]:= 16#c7c2;
    GB2312[6104]:= 16#eff1;
    GB2312[6105]:= 16#b6cd;
    GB2312[6106]:= 16#efcb;
    GB2312[6107]:= 16#efcc;
    GB2312[6108]:= 16#efcd;
    GB2312[6109]:= 16#b6c6;
    GB2312[6110]:= 16#c3be;
    GB2312[6111]:= 16#efce;
    GB2312[6112]:= 16#efd0;
    GB2312[6113]:= 16#efd1;
    GB2312[6114]:= 16#efd2;
    GB2312[6115]:= 16#d5f2;
    GB2312[6116]:= 16#efd3;
    GB2312[6117]:= 16#c4f7;
    GB2312[6118]:= 16#efd4;
    GB2312[6119]:= 16#c4f8;
    GB2312[6120]:= 16#efd5;
    GB2312[6121]:= 16#efd6;
    GB2312[6122]:= 16#b8e4;
    GB2312[6123]:= 16#b0f7;
    GB2312[6124]:= 16#efd7;
    GB2312[6125]:= 16#efd8;
    GB2312[6126]:= 16#efd9;
    GB2312[6127]:= 16#efda;
    GB2312[6128]:= 16#efdb;
    GB2312[6129]:= 16#efdc;
    GB2312[6130]:= 16#efdd;
    GB2312[6131]:= 16#efde;
    GB2312[6132]:= 16#beb5;
    GB2312[6133]:= 16#efe1;
    GB2312[6134]:= 16#efdf;
    GB2312[6135]:= 16#efe0;
    GB2312[6136]:= 16#efe2;
    GB2312[6137]:= 16#efe3;
    GB2312[6138]:= 16#c1cd;
    GB2312[6139]:= 16#efe4;
    GB2312[6140]:= 16#efe5;
    GB2312[6141]:= 16#efe6;
    GB2312[6142]:= 16#efe7;
    GB2312[6143]:= 16#efe8;
    GB2312[6144]:= 16#efe9;
    GB2312[6145]:= 16#efea;
    GB2312[6146]:= 16#efeb;
    GB2312[6147]:= 16#efec;
    GB2312[6148]:= 16#c0d8;
    GB2312[6149]:= 16#efed;
    GB2312[6150]:= 16#c1ad;
    GB2312[6151]:= 16#efee;
    GB2312[6152]:= 16#efef;
    GB2312[6153]:= 16#eff0;
    GB2312[6154]:= 16#cfe2;
    GB2312[6155]:= 16#b3a4;
    GB2312[6156]:= 16#c3c5;
    GB2312[6157]:= 16#e3c5;
    GB2312[6158]:= 16#c9c1;
    GB2312[6159]:= 16#e3c6;
    GB2312[6160]:= 16#b1d5;
    GB2312[6161]:= 16#ceca;
    GB2312[6162]:= 16#b4b3;
    GB2312[6163]:= 16#c8f2;
    GB2312[6164]:= 16#e3c7;
    GB2312[6165]:= 16#cfd0;
    GB2312[6166]:= 16#e3c8;
    GB2312[6167]:= 16#bce4;
    GB2312[6168]:= 16#e3c9;
    GB2312[6169]:= 16#e3ca;
    GB2312[6170]:= 16#c3c6;
    GB2312[6171]:= 16#d5a2;
    GB2312[6172]:= 16#c4d6;
    GB2312[6173]:= 16#b9eb;
    GB2312[6174]:= 16#cec5;
    GB2312[6175]:= 16#e3cb;
    GB2312[6176]:= 16#c3f6;
    GB2312[6177]:= 16#e3cc;
    GB2312[6178]:= 16#b7a7;
    GB2312[6179]:= 16#b8f3;
    GB2312[6180]:= 16#bad2;
    GB2312[6181]:= 16#e3cd;
    GB2312[6182]:= 16#e3ce;
    GB2312[6183]:= 16#d4c4;
    GB2312[6184]:= 16#e3cf;
    GB2312[6185]:= 16#e3d0;
    GB2312[6186]:= 16#d1cb;
    GB2312[6187]:= 16#e3d1;
    GB2312[6188]:= 16#e3d2;
    GB2312[6189]:= 16#e3d3;
    GB2312[6190]:= 16#e3d4;
    GB2312[6191]:= 16#d1d6;
    GB2312[6192]:= 16#e3d5;
    GB2312[6193]:= 16#b2fb;
    GB2312[6194]:= 16#c0bb;
    GB2312[6195]:= 16#e3d6;
    GB2312[6196]:= 16#c0ab;
    GB2312[6197]:= 16#e3d7;
    GB2312[6198]:= 16#e3d8;
    GB2312[6199]:= 16#e3d9;
    GB2312[6200]:= 16#e3da;
    GB2312[6201]:= 16#e3db;
    GB2312[6202]:= 16#b8b7;
    GB2312[6203]:= 16#dae2;
    GB2312[6204]:= 16#b6d3;
    GB2312[6205]:= 16#dae4;
    GB2312[6206]:= 16#dae3;
    GB2312[6207]:= 16#dae6;
    GB2312[6208]:= 16#c8ee;
    GB2312[6209]:= 16#dae5;
    GB2312[6210]:= 16#b7c0;
    GB2312[6211]:= 16#d1f4;
    GB2312[6212]:= 16#d2f5;
    GB2312[6213]:= 16#d5f3;
    GB2312[6214]:= 16#bdd7;
    GB2312[6215]:= 16#d7e8;
    GB2312[6216]:= 16#dae8;
    GB2312[6217]:= 16#dae7;
    GB2312[6218]:= 16#b0a2;
    GB2312[6219]:= 16#cdd3;
    GB2312[6220]:= 16#dae9;
    GB2312[6221]:= 16#b8bd;
    GB2312[6222]:= 16#bcca;
    GB2312[6223]:= 16#c2bd;
    GB2312[6224]:= 16#c2a4;
    GB2312[6225]:= 16#b3c2;
    GB2312[6226]:= 16#daea;
    GB2312[6227]:= 16#c2aa;
    GB2312[6228]:= 16#c4b0;
    GB2312[6229]:= 16#bdb5;
    GB2312[6230]:= 16#cfde;
    GB2312[6231]:= 16#daeb;
    GB2312[6232]:= 16#c9c2;
    GB2312[6233]:= 16#b1dd;
    GB2312[6234]:= 16#daec;
    GB2312[6235]:= 16#b6b8;
    GB2312[6236]:= 16#d4ba;
    GB2312[6237]:= 16#b3fd;
    GB2312[6238]:= 16#daed;
    GB2312[6239]:= 16#d4c9;
    GB2312[6240]:= 16#cfd5;
    GB2312[6241]:= 16#c5e3;
    GB2312[6242]:= 16#daee;
    GB2312[6243]:= 16#daef;
    GB2312[6244]:= 16#daf0;
    GB2312[6245]:= 16#c1ea;
    GB2312[6246]:= 16#ccd5;
    GB2312[6247]:= 16#cfdd;
    GB2312[6248]:= 16#d3e7;
    GB2312[6249]:= 16#c2a1;
    GB2312[6250]:= 16#daf1;
    GB2312[6251]:= 16#cbe5;
    GB2312[6252]:= 16#daf2;
    GB2312[6253]:= 16#cbe6;
    GB2312[6254]:= 16#d2fe;
    GB2312[6255]:= 16#b8f4;
    GB2312[6256]:= 16#daf3;
    GB2312[6257]:= 16#b0af;
    GB2312[6258]:= 16#cfb6;
    GB2312[6259]:= 16#d5cf;
    GB2312[6260]:= 16#cbed;
    GB2312[6261]:= 16#daf4;
    GB2312[6262]:= 16#e3c4;
    GB2312[6263]:= 16#c1a5;
    GB2312[6264]:= 16#f6bf;
    GB2312[6265]:= 16#f6c0;
    GB2312[6266]:= 16#f6c1;
    GB2312[6267]:= 16#c4d1;
    GB2312[6268]:= 16#c8b8;
    GB2312[6269]:= 16#d1e3;
    GB2312[6270]:= 16#d0db;
    GB2312[6271]:= 16#d1c5;
    GB2312[6272]:= 16#bcaf;
    GB2312[6273]:= 16#b9cd;
    GB2312[6274]:= 16#eff4;
    GB2312[6275]:= 16#b4c6;
    GB2312[6276]:= 16#d3ba;
    GB2312[6277]:= 16#f6c2;
    GB2312[6278]:= 16#b3fb;
    GB2312[6279]:= 16#f6c3;
    GB2312[6280]:= 16#b5f1;
    GB2312[6281]:= 16#f6c5;
    GB2312[6282]:= 16#d3ea;
    GB2312[6283]:= 16#f6a7;
    GB2312[6284]:= 16#d1a9;
    GB2312[6285]:= 16#f6a9;
    GB2312[6286]:= 16#f6a8;
    GB2312[6287]:= 16#c1e3;
    GB2312[6288]:= 16#c0d7;
    GB2312[6289]:= 16#b1a2;
    GB2312[6290]:= 16#ceed;
    GB2312[6291]:= 16#d0e8;
    GB2312[6292]:= 16#f6ab;
    GB2312[6293]:= 16#cff6;
    GB2312[6294]:= 16#f6aa;
    GB2312[6295]:= 16#d5f0;
    GB2312[6296]:= 16#f6ac;
    GB2312[6297]:= 16#c3b9;
    GB2312[6298]:= 16#bbf4;
    GB2312[6299]:= 16#f6ae;
    GB2312[6300]:= 16#f6ad;
    GB2312[6301]:= 16#c4de;
    GB2312[6302]:= 16#c1d8;
    GB2312[6303]:= 16#cbaa;
    GB2312[6304]:= 16#cfbc;
    GB2312[6305]:= 16#f6af;
    GB2312[6306]:= 16#f6b0;
    GB2312[6307]:= 16#f6b1;
    GB2312[6308]:= 16#c2b6;
    GB2312[6309]:= 16#b0d4;
    GB2312[6310]:= 16#c5f9;
    GB2312[6311]:= 16#f6b2;
    GB2312[6312]:= 16#c7e0;
    GB2312[6313]:= 16#f6a6;
    GB2312[6314]:= 16#beb8;
    GB2312[6315]:= 16#beb2;
    GB2312[6316]:= 16#b5e5;
    GB2312[6317]:= 16#b7c7;
    GB2312[6318]:= 16#bfbf;
    GB2312[6319]:= 16#c3d2;
    GB2312[6320]:= 16#c3e6;
    GB2312[6321]:= 16#d8cc;
    GB2312[6322]:= 16#b8ef;
    GB2312[6323]:= 16#bdf9;
    GB2312[6324]:= 16#d1a5;
    GB2312[6325]:= 16#b0d0;
    GB2312[6326]:= 16#f7b0;
    GB2312[6327]:= 16#f7b1;
    GB2312[6328]:= 16#d0ac;
    GB2312[6329]:= 16#b0b0;
    GB2312[6330]:= 16#f7b2;
    GB2312[6331]:= 16#f7b3;
    GB2312[6332]:= 16#f7b4;
    GB2312[6333]:= 16#c7ca;
    GB2312[6334]:= 16#becf;
    GB2312[6335]:= 16#f7b7;
    GB2312[6336]:= 16#f7b6;
    GB2312[6337]:= 16#b1de;
    GB2312[6338]:= 16#f7b5;
    GB2312[6339]:= 16#f7b8;
    GB2312[6340]:= 16#f7b9;
    GB2312[6341]:= 16#cea4;
    GB2312[6342]:= 16#c8cd;
    GB2312[6343]:= 16#baab;
    GB2312[6344]:= 16#e8b8;
    GB2312[6345]:= 16#e8b9;
    GB2312[6346]:= 16#e8ba;
    GB2312[6347]:= 16#bec2;
    GB2312[6348]:= 16#d2f4;
    GB2312[6349]:= 16#d4cf;
    GB2312[6350]:= 16#c9d8;
    GB2312[6351]:= 16#d2b3;
    GB2312[6352]:= 16#b6a5;
    GB2312[6353]:= 16#c7ea;
    GB2312[6354]:= 16#f1fc;
    GB2312[6355]:= 16#cfee;
    GB2312[6356]:= 16#cbb3;
    GB2312[6357]:= 16#d0eb;
    GB2312[6358]:= 16#e7ef;
    GB2312[6359]:= 16#cde7;
    GB2312[6360]:= 16#b9cb;
    GB2312[6361]:= 16#b6d9;
    GB2312[6362]:= 16#f1fd;
    GB2312[6363]:= 16#b0e4;
    GB2312[6364]:= 16#cbcc;
    GB2312[6365]:= 16#f1fe;
    GB2312[6366]:= 16#d4a4;
    GB2312[6367]:= 16#c2ad;
    GB2312[6368]:= 16#c1ec;
    GB2312[6369]:= 16#c6c4;
    GB2312[6370]:= 16#beb1;
    GB2312[6371]:= 16#f2a1;
    GB2312[6372]:= 16#bcd5;
    GB2312[6373]:= 16#f2a2;
    GB2312[6374]:= 16#f2a3;
    GB2312[6375]:= 16#f2a4;
    GB2312[6376]:= 16#d2c3;
    GB2312[6377]:= 16#c6b5;
    GB2312[6378]:= 16#cdc7;
    GB2312[6379]:= 16#f2a5;
    GB2312[6380]:= 16#d3b1;
    GB2312[6381]:= 16#bfc5;
    GB2312[6382]:= 16#cce2;
    GB2312[6383]:= 16#f2a6;
    GB2312[6384]:= 16#f2a7;
    GB2312[6385]:= 16#d1d5;
    GB2312[6386]:= 16#b6ee;
    GB2312[6387]:= 16#f2a8;
    GB2312[6388]:= 16#f2a9;
    GB2312[6389]:= 16#b5df;
    GB2312[6390]:= 16#f2aa;
    GB2312[6391]:= 16#f2ab;
    GB2312[6392]:= 16#b2fc;
    GB2312[6393]:= 16#f2ac;
    GB2312[6394]:= 16#f2ad;
    GB2312[6395]:= 16#c8a7;
    GB2312[6396]:= 16#b7e7;
    GB2312[6397]:= 16#eca9;
    GB2312[6398]:= 16#ecaa;
    GB2312[6399]:= 16#ecab;
    GB2312[6400]:= 16#ecac;
    GB2312[6401]:= 16#c6ae;
    GB2312[6402]:= 16#ecad;
    GB2312[6403]:= 16#ecae;
    GB2312[6404]:= 16#b7c9;
    GB2312[6405]:= 16#cab3;
    GB2312[6406]:= 16#e2b8;
    GB2312[6407]:= 16#f7cf;
    GB2312[6408]:= 16#f7d0;
    GB2312[6409]:= 16#b2cd;
    GB2312[6410]:= 16#f7d1;
    GB2312[6411]:= 16#f7d3;
    GB2312[6412]:= 16#f7d2;
    GB2312[6413]:= 16#e2bb;
    GB2312[6414]:= 16#bca2;
    GB2312[6415]:= 16#e2bc;
    GB2312[6416]:= 16#e2bd;
    GB2312[6417]:= 16#e2be;
    GB2312[6418]:= 16#e2bf;
    GB2312[6419]:= 16#e2c0;
    GB2312[6420]:= 16#e2c1;
    GB2312[6421]:= 16#b7b9;
    GB2312[6422]:= 16#d2fb;
    GB2312[6423]:= 16#bda4;
    GB2312[6424]:= 16#cace;
    GB2312[6425]:= 16#b1a5;
    GB2312[6426]:= 16#cbc7;
    GB2312[6427]:= 16#e2c2;
    GB2312[6428]:= 16#b6fc;
    GB2312[6429]:= 16#c8c4;
    GB2312[6430]:= 16#e2c3;
    GB2312[6431]:= 16#bdc8;
    GB2312[6432]:= 16#b1fd;
    GB2312[6433]:= 16#e2c4;
    GB2312[6434]:= 16#b6f6;
    GB2312[6435]:= 16#e2c5;
    GB2312[6436]:= 16#c4d9;
    GB2312[6437]:= 16#e2c6;
    GB2312[6438]:= 16#cfda;
    GB2312[6439]:= 16#b9dd;
    GB2312[6440]:= 16#e2c7;
    GB2312[6441]:= 16#c0a1;
    GB2312[6442]:= 16#e2c8;
    GB2312[6443]:= 16#b2f6;
    GB2312[6444]:= 16#e2c9;
    GB2312[6445]:= 16#c1f3;
    GB2312[6446]:= 16#e2ca;
    GB2312[6447]:= 16#e2cb;
    GB2312[6448]:= 16#c2f8;
    GB2312[6449]:= 16#e2cc;
    GB2312[6450]:= 16#e2cd;
    GB2312[6451]:= 16#e2ce;
    GB2312[6452]:= 16#cad7;
    GB2312[6453]:= 16#d8b8;
    GB2312[6454]:= 16#d9e5;
    GB2312[6455]:= 16#cfe3;
    GB2312[6456]:= 16#f0a5;
    GB2312[6457]:= 16#dcb0;
    GB2312[6458]:= 16#c2ed;
    GB2312[6459]:= 16#d4a6;
    GB2312[6460]:= 16#cdd4;
    GB2312[6461]:= 16#d1b1;
    GB2312[6462]:= 16#b3db;
    GB2312[6463]:= 16#c7fd;
    GB2312[6464]:= 16#b2b5;
    GB2312[6465]:= 16#c2bf;
    GB2312[6466]:= 16#e6e0;
    GB2312[6467]:= 16#cabb;
    GB2312[6468]:= 16#e6e1;
    GB2312[6469]:= 16#e6e2;
    GB2312[6470]:= 16#bed4;
    GB2312[6471]:= 16#e6e3;
    GB2312[6472]:= 16#d7a4;
    GB2312[6473]:= 16#cdd5;
    GB2312[6474]:= 16#e6e5;
    GB2312[6475]:= 16#bcdd;
    GB2312[6476]:= 16#e6e4;
    GB2312[6477]:= 16#e6e6;
    GB2312[6478]:= 16#e6e7;
    GB2312[6479]:= 16#c2ee;
    GB2312[6480]:= 16#bdbe;
    GB2312[6481]:= 16#e6e8;
    GB2312[6482]:= 16#c2e6;
    GB2312[6483]:= 16#baa7;
    GB2312[6484]:= 16#e6e9;
    GB2312[6485]:= 16#e6ea;
    GB2312[6486]:= 16#b3d2;
    GB2312[6487]:= 16#d1e9;
    GB2312[6488]:= 16#bfa5;
    GB2312[6489]:= 16#e6eb;
    GB2312[6490]:= 16#c6ef;
    GB2312[6491]:= 16#e6ec;
    GB2312[6492]:= 16#e6ed;
    GB2312[6493]:= 16#e6ee;
    GB2312[6494]:= 16#c6ad;
    GB2312[6495]:= 16#e6ef;
    GB2312[6496]:= 16#c9a7;
    GB2312[6497]:= 16#e6f0;
    GB2312[6498]:= 16#e6f1;
    GB2312[6499]:= 16#e6f2;
    GB2312[6500]:= 16#e5b9;
    GB2312[6501]:= 16#e6f3;
    GB2312[6502]:= 16#e6f4;
    GB2312[6503]:= 16#c2e2;
    GB2312[6504]:= 16#e6f5;
    GB2312[6505]:= 16#e6f6;
    GB2312[6506]:= 16#d6e8;
    GB2312[6507]:= 16#e6f7;
    GB2312[6508]:= 16#e6f8;
    GB2312[6509]:= 16#b9c7;
    GB2312[6510]:= 16#f7bb;
    GB2312[6511]:= 16#f7ba;
    GB2312[6512]:= 16#f7be;
    GB2312[6513]:= 16#f7bc;
    GB2312[6514]:= 16#baa1;
    GB2312[6515]:= 16#f7bf;
    GB2312[6516]:= 16#f7c0;
    GB2312[6517]:= 16#f7c2;
    GB2312[6518]:= 16#f7c1;
    GB2312[6519]:= 16#f7c4;
    GB2312[6520]:= 16#f7c3;
    GB2312[6521]:= 16#f7c5;
    GB2312[6522]:= 16#f7c6;
    GB2312[6523]:= 16#f7c7;
    GB2312[6524]:= 16#cbe8;
    GB2312[6525]:= 16#b8df;
    GB2312[6526]:= 16#f7d4;
    GB2312[6527]:= 16#f7d5;
    GB2312[6528]:= 16#f7d6;
    GB2312[6529]:= 16#f7d8;
    GB2312[6530]:= 16#f7da;
    GB2312[6531]:= 16#f7d7;
    GB2312[6532]:= 16#f7db;
    GB2312[6533]:= 16#f7d9;
    GB2312[6534]:= 16#d7d7;
    GB2312[6535]:= 16#f7dc;
    GB2312[6536]:= 16#f7dd;
    GB2312[6537]:= 16#f7de;
    GB2312[6538]:= 16#f7df;
    GB2312[6539]:= 16#f7e0;
    GB2312[6540]:= 16#dbcb;
    GB2312[6541]:= 16#d8aa;
    GB2312[6542]:= 16#e5f7;
    GB2312[6543]:= 16#b9ed;
    GB2312[6544]:= 16#bffd;
    GB2312[6545]:= 16#bbea;
    GB2312[6546]:= 16#f7c9;
    GB2312[6547]:= 16#c6c7;
    GB2312[6548]:= 16#f7c8;
    GB2312[6549]:= 16#f7ca;
    GB2312[6550]:= 16#f7cc;
    GB2312[6551]:= 16#f7cb;
    GB2312[6552]:= 16#f7cd;
    GB2312[6553]:= 16#ceba;
    GB2312[6554]:= 16#f7ce;
    GB2312[6555]:= 16#c4a7;
    GB2312[6556]:= 16#d3e3;
    GB2312[6557]:= 16#f6cf;
    GB2312[6558]:= 16#c2b3;
    GB2312[6559]:= 16#f6d0;
    GB2312[6560]:= 16#f6d1;
    GB2312[6561]:= 16#f6d2;
    GB2312[6562]:= 16#f6d3;
    GB2312[6563]:= 16#f6d4;
    GB2312[6564]:= 16#f6d6;
    GB2312[6565]:= 16#b1ab;
    GB2312[6566]:= 16#f6d7;
    GB2312[6567]:= 16#f6d8;
    GB2312[6568]:= 16#f6d9;
    GB2312[6569]:= 16#f6da;
    GB2312[6570]:= 16#f6db;
    GB2312[6571]:= 16#f6dc;
    GB2312[6572]:= 16#f6dd;
    GB2312[6573]:= 16#f6de;
    GB2312[6574]:= 16#cfca;
    GB2312[6575]:= 16#f6df;
    GB2312[6576]:= 16#f6e0;
    GB2312[6577]:= 16#f6e1;
    GB2312[6578]:= 16#f6e2;
    GB2312[6579]:= 16#f6e3;
    GB2312[6580]:= 16#f6e4;
    GB2312[6581]:= 16#c0f0;
    GB2312[6582]:= 16#f6e5;
    GB2312[6583]:= 16#f6e6;
    GB2312[6584]:= 16#f6e7;
    GB2312[6585]:= 16#f6e8;
    GB2312[6586]:= 16#f6e9;
    GB2312[6587]:= 16#f6ea;
    GB2312[6588]:= 16#f6eb;
    GB2312[6589]:= 16#f6ec;
    GB2312[6590]:= 16#f6ed;
    GB2312[6591]:= 16#f6ee;
    GB2312[6592]:= 16#f6ef;
    GB2312[6593]:= 16#f6f0;
    GB2312[6594]:= 16#f6f1;
    GB2312[6595]:= 16#f6f2;
    GB2312[6596]:= 16#f6f3;
    GB2312[6597]:= 16#f6f4;
    GB2312[6598]:= 16#bea8;
    GB2312[6599]:= 16#f6f5;
    GB2312[6600]:= 16#f6f6;
    GB2312[6601]:= 16#f6f7;
    GB2312[6602]:= 16#f6f8;
    GB2312[6603]:= 16#c8fa;
    GB2312[6604]:= 16#f6f9;
    GB2312[6605]:= 16#f6fa;
    GB2312[6606]:= 16#f6fb;
    GB2312[6607]:= 16#f6fc;
    GB2312[6608]:= 16#f6fd;
    GB2312[6609]:= 16#f6fe;
    GB2312[6610]:= 16#f7a1;
    GB2312[6611]:= 16#f7a2;
    GB2312[6612]:= 16#f7a3;
    GB2312[6613]:= 16#f7a4;
    GB2312[6614]:= 16#f7a5;
    GB2312[6615]:= 16#f7a6;
    GB2312[6616]:= 16#f7a7;
    GB2312[6617]:= 16#f7a8;
    GB2312[6618]:= 16#b1ee;
    GB2312[6619]:= 16#f7a9;
    GB2312[6620]:= 16#f7aa;
    GB2312[6621]:= 16#f7ab;
    GB2312[6622]:= 16#f7ac;
    GB2312[6623]:= 16#f7ad;
    GB2312[6624]:= 16#c1db;
    GB2312[6625]:= 16#f7ae;
    GB2312[6626]:= 16#f7af;
    GB2312[6627]:= 16#c4f1;
    GB2312[6628]:= 16#f0af;
    GB2312[6629]:= 16#bca6;
    GB2312[6630]:= 16#f0b0;
    GB2312[6631]:= 16#c3f9;
    GB2312[6632]:= 16#c5b8;
    GB2312[6633]:= 16#d1bb;
    GB2312[6634]:= 16#f0b1;
    GB2312[6635]:= 16#f0b2;
    GB2312[6636]:= 16#f0b3;
    GB2312[6637]:= 16#f0b4;
    GB2312[6638]:= 16#f0b5;
    GB2312[6639]:= 16#d1bc;
    GB2312[6640]:= 16#d1ec;
    GB2312[6641]:= 16#f0b7;
    GB2312[6642]:= 16#f0b6;
    GB2312[6643]:= 16#d4a7;
    GB2312[6644]:= 16#cdd2;
    GB2312[6645]:= 16#f0b8;
    GB2312[6646]:= 16#f0ba;
    GB2312[6647]:= 16#f0b9;
    GB2312[6648]:= 16#f0bb;
    GB2312[6649]:= 16#f0bc;
    GB2312[6650]:= 16#b8eb;
    GB2312[6651]:= 16#f0bd;
    GB2312[6652]:= 16#bae8;
    GB2312[6653]:= 16#f0be;
    GB2312[6654]:= 16#f0bf;
    GB2312[6655]:= 16#bee9;
    GB2312[6656]:= 16#f0c0;
    GB2312[6657]:= 16#b6ec;
    GB2312[6658]:= 16#f0c1;
    GB2312[6659]:= 16#f0c2;
    GB2312[6660]:= 16#f0c3;
    GB2312[6661]:= 16#f0c4;
    GB2312[6662]:= 16#c8b5;
    GB2312[6663]:= 16#f0c5;
    GB2312[6664]:= 16#f0c6;
    GB2312[6665]:= 16#f0c7;
    GB2312[6666]:= 16#c5f4;
    GB2312[6667]:= 16#f0c8;
    GB2312[6668]:= 16#f0c9;
    GB2312[6669]:= 16#f0ca;
    GB2312[6670]:= 16#f7bd;
    GB2312[6671]:= 16#f0cb;
    GB2312[6672]:= 16#f0cc;
    GB2312[6673]:= 16#f0cd;
    GB2312[6674]:= 16#f0ce;
    GB2312[6675]:= 16#f0cf;
    GB2312[6676]:= 16#bad7;
    GB2312[6677]:= 16#f0d0;
    GB2312[6678]:= 16#f0d1;
    GB2312[6679]:= 16#f0d2;
    GB2312[6680]:= 16#f0d3;
    GB2312[6681]:= 16#f0d4;
    GB2312[6682]:= 16#f0d5;
    GB2312[6683]:= 16#f0d6;
    GB2312[6684]:= 16#f0d8;
    GB2312[6685]:= 16#d3a5;
    GB2312[6686]:= 16#f0d7;
    GB2312[6687]:= 16#f0d9;
    GB2312[6688]:= 16#f5ba;
    GB2312[6689]:= 16#c2b9;
    GB2312[6690]:= 16#f7e4;
    GB2312[6691]:= 16#f7e5;
    GB2312[6692]:= 16#f7e6;
    GB2312[6693]:= 16#f7e7;
    GB2312[6694]:= 16#f7e8;
    GB2312[6695]:= 16#c2b4;
    GB2312[6696]:= 16#f7ea;
    GB2312[6697]:= 16#f7eb;
    GB2312[6698]:= 16#c2f3;
    GB2312[6699]:= 16#f4f0;
    GB2312[6700]:= 16#f4ef;
    GB2312[6701]:= 16#c2e9;
    GB2312[6702]:= 16#f7e1;
    GB2312[6703]:= 16#f7e2;
    GB2312[6704]:= 16#bbc6;
    GB2312[6705]:= 16#d9e4;
    GB2312[6706]:= 16#caf2;
    GB2312[6707]:= 16#c0e8;
    GB2312[6708]:= 16#f0a4;
    GB2312[6709]:= 16#bada;
    GB2312[6710]:= 16#c7ad;
    GB2312[6711]:= 16#c4ac;
    GB2312[6712]:= 16#f7ec;
    GB2312[6713]:= 16#f7ed;
    GB2312[6714]:= 16#f7ee;
    GB2312[6715]:= 16#f7f0;
    GB2312[6716]:= 16#f7ef;
    GB2312[6717]:= 16#f7f1;
    GB2312[6718]:= 16#f7f4;
    GB2312[6719]:= 16#f7f3;
    GB2312[6720]:= 16#f7f2;
    GB2312[6721]:= 16#f7f5;
    GB2312[6722]:= 16#f7f6;
    GB2312[6723]:= 16#ede9;
    GB2312[6724]:= 16#edea;
    GB2312[6725]:= 16#edeb;
    GB2312[6726]:= 16#f6bc;
    GB2312[6727]:= 16#f6bd;
    GB2312[6728]:= 16#f6be;
    GB2312[6729]:= 16#b6a6;
    GB2312[6730]:= 16#d8be;
    GB2312[6731]:= 16#b9c4;
    GB2312[6732]:= 16#d8bb;
    GB2312[6733]:= 16#dcb1;
    GB2312[6734]:= 16#caf3;
    GB2312[6735]:= 16#f7f7;
    GB2312[6736]:= 16#f7f8;
    GB2312[6737]:= 16#f7f9;
    GB2312[6738]:= 16#f7fb;
    GB2312[6739]:= 16#f7fa;
    GB2312[6740]:= 16#b1c7;
    GB2312[6741]:= 16#f7fc;
    GB2312[6742]:= 16#f7fd;
    GB2312[6743]:= 16#f7fe;
    GB2312[6744]:= 16#c6eb;
    GB2312[6745]:= 16#ecb4;
    GB2312[6746]:= 16#b3dd;
    GB2312[6747]:= 16#f6b3;
    GB2312[6748]:= 16#f6b4;
    GB2312[6749]:= 16#c1e4;
    GB2312[6750]:= 16#f6b5;
    GB2312[6751]:= 16#f6b6;
    GB2312[6752]:= 16#f6b7;
    GB2312[6753]:= 16#f6b8;
    GB2312[6754]:= 16#f6b9;
    GB2312[6755]:= 16#f6ba;
    GB2312[6756]:= 16#c8a3;
    GB2312[6757]:= 16#f6bb;
    GB2312[6758]:= 16#c1fa;
    GB2312[6759]:= 16#b9a8;
    GB2312[6760]:= 16#ede8;
    GB2312[6761]:= 16#b9ea;
    GB2312[6762]:= 16#d9df;
    GB2312[6763]:= 16#d7fa;
    GB2312[6764]:= 16#d7fb;
    GB2312[6765]:= 16#d7fc;
    GB2312[6766]:= 16#d7fd;
    GB2312[6767]:= 16#d7fe;
    GB2312[6768]:= 16#a3a1;
    GB2312[6769]:= 16#a3a8;
    GB2312[6770]:= 16#a3a9;
    GB2312[6771]:= 16#a3ac;
    GB2312[6772]:= 16#a3ba;
    GB2312[6773]:= 16#a3bb;
    GB2312[6774]:= 16#a3bf;
    GB2312[6775]:= 16#a3a4;            //GB2312码 6000-6999
END_IF;
END_FUNCTION_BLOCK